LIN {X 0,Y 737.28,Z 922.886,A -85,B 0,C 180,E1 34854.05,E2 34854.05} C_VEL
LIN {X 0,Y 736.992,Z 943.234,A -85,B 0,C 180,E1 34852.747,E2 34852.747} C_VEL
LIN {X 0,Y 736.792,Z 961.106,A -85,B 0,C 180,E1 34851.449,E2 34851.449} C_VEL
LIN {X 0,Y 736.567,Z 978.603,A -85,B 0,C 180,E1 34850.004,E2 34850.004} C_VEL
LIN {X 0,Y 736.424,Z 994.494,A -85,B 0,C 180,E1 34848.525,E2 34848.525} C_VEL
LIN {X 0,Y 736.245,Z 1009.802,A -85,B 0,C 180,E1 34846.896,E2 34846.896} C_VEL
LIN {X 0,Y 736.159,Z 1022.669,A -85,B 0,C 180,E1 34845.342,E2 34845.342} C_VEL
LIN {X 0,Y 736.056,Z 1035.753,A -85,B 0,C 180,E1 34843.512,E2 34843.512} C_VEL
LIN {X 0,Y 735.988,Z 1045.128,A -85,B 0,C 180,E1 34841.993,E2 34841.993} C_VEL
LIN {X 0,Y 735.962,Z 1054.76,A -85,B 0,C 180,E1 34840.173,E2 34840.173} C_VEL
LIN {X 0,Y 735.918,Z 1062.206,A -85,B 0,C 180,E1 34838.438,E2 34838.438} C_VEL
LIN {X 0,Y 735.911,Z 1067.997,A -85,B 0,C 180,E1 34836.789,E2 34836.789} C_VEL
LIN {X 0,Y 735.917,Z 1073.178,A -85,B 0,C 180,E1 34834.832,E2 34834.832} C_VEL
LIN {X 0,Y 735.916,Z 1076.234,A -85,B 0,C 180,E1 34833.115,E2 34833.115} C_VEL
LIN {X 0,Y 735.907,Z 1078.149,A -85,B 0,C 180,E1 34831.246,E2 34831.246} C_VEL
LIN {X 0,Y 735.891,Z 1078.351,A -85,B 0,C 180,E1 34829.455,E2 34829.455} C_VEL
LIN {X 0,Y 735.914,Z 1077.297,A -85,B 0,C 180,E1 34827.742,E2 34827.742} C_VEL
LIN {X 0,Y 735.908,Z 1074.445,A -85,B 0,C 180,E1 34825.792,E2 34825.792} C_VEL
LIN {X 0,Y 735.918,Z 1070.688,A -85,B 0,C 180,E1 34824.151,E2 34824.151} C_VEL
LIN {X 0,Y 735.911,Z 1064.936,A -85,B 0,C 180,E1 34822.27,E2 34822.27} C_VEL
LIN {X 0,Y 735.931,Z 1057.601,A -85,B 0,C 180,E1 34820.459,E2 34820.459} C_VEL
LIN {X 0,Y 735.974,Z 1049.926,A -85,B 0,C 180,E1 34818.877,E2 34818.877} C_VEL
LIN {X 0,Y 736.039,Z 1038.526,A -85,B 0,C 180,E1 34816.914,E2 34816.914} C_VEL
LIN {X 0,Y 736.104,Z 1027.954,A -85,B 0,C 180,E1 34815.365,E2 34815.365} C_VEL
LIN {X 0,Y 736.23,Z 1014.045,A -85,B 0,C 180,E1 34813.591,E2 34813.591} C_VEL
LIN {X 0,Y 736.33,Z 1000.068,A -85,B 0,C 180,E1 34812.046,E2 34812.046} C_VEL
LIN {X 0,Y 736.542,Z 983.248,A -85,B 0,C 180,E1 34810.408,E2 34810.408} C_VEL
LIN {X 0,Y 736.708,Z 966.807,A -85,B 0,C 180,E1 34809.003,E2 34809.003} C_VEL
LIN {X 0,Y 736.965,Z 946.856,A -85,B 0,C 180,E1 34807.505,E2 34807.505} C_VEL
LIN {X 0,Y 737.196,Z 928.356,A -85,B 0,C 180,E1 34806.282,E2 34806.282} C_VEL
LIN {X 0,Y 737.48,Z 906.347,A -85,B 0,C 180,E1 34805.018,E2 34805.018} C_VEL
LIN {X 0,Y 737.719,Z 886.789,A -85,B 0,C 180,E1 34804.037,E2 34804.037} C_VEL
LIN {X 0,Y 738.022,Z 863.387,A -85,B 0,C 180,E1 34803.034,E2 34803.034} C_VEL
LIN {X 0,Y 738.198,Z 843.697,A -85,B 0,C 180,E1 34802.316,E2 34802.316} C_VEL
LIN {X 0,Y 738.494,Z 820.044,A -85,B 0,C 180,E1 34801.595,E2 34801.595} C_VEL
LIN {X 0,Y 738.641,Z 797.319,A -85,B 0,C 180,E1 34801.051,E2 34801.051} C_VEL
LIN {X 0,Y 738.792,Z 776.074,A -85,B 0,C 180,E1 34800.656,E2 34800.656} C_VEL
LIN {X 0,Y 738.933,Z 744.92,A -85,B 0,C 180,E1 34800.262,E2 34800.262} C_VEL
LIN {X 0,Y 739.5,Z 493.491,A -85,B 0,C 180,E1 34797.493,E2 34797.493} C_VEL
LIN {X 0,Y 739.604,Z 381.804,A -85,B 0,C 180,E1 34796.229,E2 34796.229} C_VEL
LIN {X 0,Y 738.409,Z 376.685,A -85,B 0,C 180,E1 34796.09,E2 34796.09} C_VEL
LIN {X 0,Y 738.712,Z 341.298,A -85,B 0,C 180,E1 34793.646,E2 34793.646} C_VEL
LIN {X 0,Y 738.481,Z 336.305,A -85,B 0,C 180,E1 34793.28,E2 34793.28} C_VEL
LIN {X 0,Y 736.045,Z 329.548,A -85,B 0,C 180,E1 34792.627,E2 34792.627} C_VEL
LIN {X 0,Y 736.024,Z 329.546,A -85,B 0,C 180,E1 34790.118,E2 34790.118} C_VEL
LIN {X 0,Y 736.063,Z 329.539,A -85,B 0,C 180,E1 34787.53,E2 34787.53} C_VEL
LIN {X 0,Y 736.046,Z 329.544,A -85,B 0,C 180,E1 34784.505,E2 34784.505} C_VEL
LIN {X 0,Y 736.024,Z 329.541,A -85,B 0,C 180,E1 34781.943,E2 34781.943} C_VEL
LIN {X 0,Y 736.082,Z 329.536,A -85,B 0,C 180,E1 34779.26,E2 34779.26} C_VEL
LIN {X 0,Y 736.042,Z 329.543,A -85,B 0,C 180,E1 34776.32,E2 34776.32} C_VEL
LIN {X 0,Y 736.026,Z 329.539,A -85,B 0,C 180,E1 34773.754,E2 34773.754} C_VEL
LIN {X 0,Y 736.099,Z 329.536,A -85,B 0,C 180,E1 34770.986,E2 34770.986} C_VEL
LIN {X 0,Y 736.038,Z 329.54,A -85,B 0,C 180,E1 34768.125,E2 34768.125} C_VEL
LIN {X 0,Y 736.028,Z 329.539,A -85,B 0,C 180,E1 34765.595,E2 34765.595} C_VEL
LIN {X 0,Y 736.1,Z 329.534,A -85,B 0,C 180,E1 34762.861,E2 34762.861} C_VEL
LIN {X 0,Y 736.034,Z 329.54,A -85,B 0,C 180,E1 34759.937,E2 34759.937} C_VEL
LIN {X 0,Y 736.031,Z 329.539,A -85,B 0,C 180,E1 34757.39,E2 34757.39} C_VEL
LIN {X 0,Y 736.099,Z 329.539,A -85,B 0,C 180,E1 34754.554,E2 34754.554} C_VEL
LIN {X 0,Y 736.033,Z 329.541,A -85,B 0,C 180,E1 34751.758,E2 34751.758} C_VEL
LIN {X 0,Y 736.033,Z 329.536,A -85,B 0,C 180,E1 34749.224,E2 34749.224} C_VEL
LIN {X 0,Y 736.1,Z 329.54,A -85,B 0,C 180,E1 34746.395,E2 34746.395} C_VEL
LIN {X 0,Y 736.032,Z 329.54,A -85,B 0,C 180,E1 34743.583,E2 34743.583} C_VEL
LIN {X 0,Y 736.037,Z 329.538,A -85,B 0,C 180,E1 34741.029,E2 34741.029} C_VEL
LIN {X 0,Y 736.097,Z 329.54,A -85,B 0,C 180,E1 34738.132,E2 34738.132} C_VEL
LIN {X 0,Y 736.03,Z 329.54,A -85,B 0,C 180,E1 34735.403,E2 34735.403} C_VEL
LIN {X 0,Y 736.037,Z 329.537,A -85,B 0,C 180,E1 34732.899,E2 34732.899} C_VEL
LIN {X 0,Y 736.097,Z 329.543,A -85,B 0,C 180,E1 34729.987,E2 34729.987} C_VEL
LIN {X 0,Y 736.028,Z 329.537,A -85,B 0,C 180,E1 34729.196,E2 34729.196} C_VEL
LIN {X 0,Y 735.028,Z 329.666,A -85,B 0,C 180,E1 34728.597,E2 34728.597} C_VEL
LIN {X 0,Y 728.625,Z 330.464,A -85,B 0,C 180,E1 34726.917,E2 34726.917} C_VEL
LIN {X 0,Y 728.13,Z 330.525,A -85,B 0,C 180,E1 34726.481,E2 34726.481} C_VEL
LIN {X 0,Y 728.109,Z 330.53,A -85,B 0,C 180,E1 34723.444,E2 34723.444} C_VEL
LIN {X 0,Y 728.092,Z 330.528,A -85,B 0,C 180,E1 34720.839,E2 34720.839} C_VEL
LIN {X 0,Y 728.159,Z 330.523,A -85,B 0,C 180,E1 34718.068,E2 34718.068} C_VEL
LIN {X 0,Y 728.097,Z 330.527,A -85,B 0,C 180,E1 34715.151,E2 34715.151} C_VEL
LIN {X 0,Y 728.096,Z 330.528,A -85,B 0,C 180,E1 34712.609,E2 34712.609} C_VEL
LIN {X 0,Y 728.16,Z 330.527,A -85,B 0,C 180,E1 34709.738,E2 34709.738} C_VEL
LIN {X 0,Y 728.093,Z 330.527,A -85,B 0,C 180,E1 34706.899,E2 34706.899} C_VEL
LIN {X 0,Y 728.11,Z 330.527,A -85,B 0,C 180,E1 34704.293,E2 34704.293} C_VEL
LIN {X 0,Y 728.13,Z 330.532,A -85,B 0,C 180,E1 34701.23,E2 34701.23} C_VEL
LIN {X 0,Y 728.092,Z 330.53,A -85,B 0,C 180,E1 34698.552,E2 34698.552} C_VEL
LIN {X 0,Y 728.156,Z 330.519,A -85,B 0,C 180,E1 34695.767,E2 34695.767} C_VEL
LIN {X 0,Y 728.104,Z 330.53,A -85,B 0,C 180,E1 34692.826,E2 34692.826} C_VEL
LIN {X 0,Y 728.099,Z 330.529,A -85,B 0,C 180,E1 34690.222,E2 34690.222} C_VEL
LIN {X 0,Y 728.161,Z 330.532,A -85,B 0,C 180,E1 34687.338,E2 34687.338} C_VEL
LIN {X 0,Y 728.095,Z 330.536,A -85,B 0,C 180,E1 34684.515,E2 34684.515} C_VEL
LIN {X 0,Y 728.157,Z 330.634,A -85,B 0,C 180,E1 34683.663,E2 34683.663} C_VEL
LIN {X 0,Y 731.175,Z 340.419,A -85,B 0,C 180,E1 34682.752,E2 34682.752} C_VEL
LIN {X 0,Y 731.211,Z 347.847,A -85,B 0,C 180,E1 34682.212,E2 34682.212} C_VEL
LIN {X 0,Y 733.078,Z 355.743,A -85,B 0,C 180,E1 34682.022,E2 34682.022} C_VEL
LIN {X 0,Y 732.35,Z 591.479,A -85,B 0,C 180,E1 34679.367,E2 34679.367} C_VEL
LIN {X 0,Y 731.891,Z 736.674,A -85,B 0,C 180,E1 34677.744,E2 34677.744} C_VEL
LIN {X 0,Y 731.635,Z 762.056,A -85,B 0,C 180,E1 34677.321,E2 34677.321} C_VEL
LIN {X 0,Y 731.419,Z 783.723,A -85,B 0,C 180,E1 34676.824,E2 34676.824} C_VEL
LIN {X 0,Y 731.163,Z 806.722,A -85,B 0,C 180,E1 34676.17,E2 34676.17} C_VEL
LIN {X 0,Y 730.791,Z 829.655,A -85,B 0,C 180,E1 34675.357,E2 34675.357} C_VEL
LIN {X 0,Y 730.482,Z 852.136,A -85,B 0,C 180,E1 34674.417,E2 34674.417} C_VEL
LIN {X 0,Y 730.067,Z 873.566,A -85,B 0,C 180,E1 34673.359,E2 34673.359} C_VEL
LIN {X 0,Y 729.754,Z 893.71,A -85,B 0,C 180,E1 34672.22,E2 34672.22} C_VEL
LIN {X 0,Y 729.388,Z 913.66,A -85,B 0,C 180,E1 34670.923,E2 34670.923} C_VEL
LIN {X 0,Y 729.096,Z 932.306,A -85,B 0,C 180,E1 34669.55,E2 34669.55} C_VEL
LIN {X 0,Y 728.785,Z 949.92,A -85,B 0,C 180,E1 34668.063,E2 34668.063} C_VEL
LIN {X 0,Y 728.585,Z 966.339,A -85,B 0,C 180,E1 34666.504,E2 34666.504} C_VEL
LIN {X 0,Y 728.356,Z 981.216,A -85,B 0,C 180,E1 34664.875,E2 34664.875} C_VEL
LIN {X 0,Y 728.216,Z 994.942,A -85,B 0,C 180,E1 34663.175,E2 34663.175} C_VEL
LIN {X 0,Y 728.096,Z 1006.602,A -85,B 0,C 180,E1 34661.486,E2 34661.486} C_VEL
LIN {X 0,Y 728.022,Z 1016.711,A -85,B 0,C 180,E1 34659.806,E2 34659.806} C_VEL
LIN {X 0,Y 727.951,Z 1026.298,A -85,B 0,C 180,E1 34657.895,E2 34657.895} C_VEL
LIN {X 0,Y 727.932,Z 1032.884,A -85,B 0,C 180,E1 34656.309,E2 34656.309} C_VEL
LIN {X 0,Y 727.913,Z 1039.273,A -85,B 0,C 180,E1 34654.412,E2 34654.412} C_VEL
LIN {X 0,Y 727.914,Z 1043.665,A -85,B 0,C 180,E1 34652.598,E2 34652.598} C_VEL
LIN {X 0,Y 727.906,Z 1046.575,A -85,B 0,C 180,E1 34650.866,E2 34650.866} C_VEL
LIN {X 0,Y 727.904,Z 1048.262,A -85,B 0,C 180,E1 34648.819,E2 34648.819} C_VEL
LIN {X 0,Y 727.9,Z 1048.283,A -85,B 0,C 180,E1 34647.165,E2 34647.165} C_VEL
LIN {X 0,Y 727.897,Z 1046.788,A -85,B 0,C 180,E1 34645.193,E2 34645.193} C_VEL
LIN {X 0,Y 727.916,Z 1043.949,A -85,B 0,C 180,E1 34643.453,E2 34643.453} C_VEL
LIN {X 0,Y 727.917,Z 1039.818,A -85,B 0,C 180,E1 34641.707,E2 34641.707} C_VEL
LIN {X 0,Y 727.938,Z 1033.314,A -85,B 0,C 180,E1 34639.714,E2 34639.714} C_VEL
LIN {X 0,Y 727.949,Z 1026.72,A -85,B 0,C 180,E1 34638.11,E2 34638.11} C_VEL
LIN {X 0,Y 728.024,Z 1018.026,A -85,B 0,C 180,E1 34636.336,E2 34636.336} C_VEL
LIN {X 0,Y 728.091,Z 1007.401,A -85,B 0,C 180,E1 34634.549,E2 34634.549} C_VEL
LIN {X 0,Y 728.196,Z 995.974,A -85,B 0,C 180,E1 34632.879,E2 34632.879} C_VEL
LIN {X 0,Y 728.355,Z 982.459,A -85,B 0,C 180,E1 34631.179,E2 34631.179} C_VEL
LIN {X 0,Y 728.531,Z 968.364,A -85,B 0,C 180,E1 34629.62,E2 34629.62} C_VEL
LIN {X 0,Y 728.763,Z 951.659,A -85,B 0,C 180,E1 34628.002,E2 34628.002} C_VEL
LIN {X 0,Y 729.047,Z 934.836,A -85,B 0,C 180,E1 34626.563,E2 34626.563} C_VEL
LIN {X 0,Y 729.341,Z 916.302,A -85,B 0,C 180,E1 34625.172,E2 34625.172} C_VEL
LIN {X 0,Y 729.671,Z 898.222,A -85,B 0,C 180,E1 34623.969,E2 34623.969} C_VEL
LIN {X 0,Y 730.026,Z 877.05,A -85,B 0,C 180,E1 34622.738,E2 34622.738} C_VEL
LIN {X 0,Y 730.364,Z 857.102,A -85,B 0,C 180,E1 34621.726,E2 34621.726} C_VEL
LIN {X 0,Y 730.753,Z 833.775,A -85,B 0,C 180,E1 34620.714,E2 34620.714} C_VEL
LIN {X 0,Y 731.015,Z 812.586,A -85,B 0,C 180,E1 34619.936,E2 34619.936} C_VEL
LIN {X 0,Y 731.403,Z 787.347,A -85,B 0,C 180,E1 34619.179,E2 34619.179} C_VEL
LIN {X 0,Y 731.608,Z 765.993,A -85,B 0,C 180,E1 34618.672,E2 34618.672} C_VEL
LIN {X 0,Y 731.866,Z 742.201,A -85,B 0,C 180,E1 34618.239,E2 34618.239} C_VEL
LIN {X 0,Y 732.018,Z 702.478,A -85,B 0,C 180,E1 34617.769,E2 34617.769} C_VEL
LIN {X 0,Y 732.808,Z 447.857,A -85,B 0,C 180,E1 34614.935,E2 34614.935} C_VEL
LIN {X 0,Y 732.898,Z 354.153,A -85,B 0,C 180,E1 34613.86,E2 34613.86} C_VEL
LIN {X 0,Y 731.135,Z 347.503,A -85,B 0,C 180,E1 34613.689,E2 34613.689} C_VEL
LIN {X 0,Y 731.178,Z 339.723,A -85,B 0,C 180,E1 34613.106,E2 34613.106} C_VEL
LIN {X 0,Y 728.14,Z 330.532,A -85,B 0,C 180,E1 34612.233,E2 34612.233} C_VEL
LIN {X 0,Y 728.09,Z 330.532,A -85,B 0,C 180,E1 34609.536,E2 34609.536} C_VEL
LIN {X 0,Y 728.135,Z 330.533,A -85,B 0,C 180,E1 34606.854,E2 34606.854} C_VEL
LIN {X 0,Y 728.111,Z 330.526,A -85,B 0,C 180,E1 34603.866,E2 34603.866} C_VEL
LIN {X 0,Y 728.09,Z 330.528,A -85,B 0,C 180,E1 34601.306,E2 34601.306} C_VEL
LIN {X 0,Y 728.154,Z 330.532,A -85,B 0,C 180,E1 34598.567,E2 34598.567} C_VEL
LIN {X 0,Y 728.101,Z 330.52,A -85,B 0,C 180,E1 34595.611,E2 34595.611} C_VEL
LIN {X 0,Y 728.094,Z 330.53,A -85,B 0,C 180,E1 34593.038,E2 34593.038} C_VEL
LIN {X 0,Y 728.161,Z 330.528,A -85,B 0,C 180,E1 34590.171,E2 34590.171} C_VEL
LIN {X 0,Y 728.096,Z 330.528,A -85,B 0,C 180,E1 34587.391,E2 34587.391} C_VEL
LIN {X 0,Y 728.098,Z 330.529,A -85,B 0,C 180,E1 34584.805,E2 34584.805} C_VEL
LIN {X 0,Y 728.153,Z 330.523,A -85,B 0,C 180,E1 34581.833,E2 34581.833} C_VEL
LIN {X 0,Y 728.089,Z 330.529,A -85,B 0,C 180,E1 34579.078,E2 34579.078} C_VEL
LIN {X 0,Y 728.121,Z 330.531,A -85,B 0,C 180,E1 34576.433,E2 34576.433} C_VEL
LIN {X 0,Y 728.117,Z 330.525,A -85,B 0,C 180,E1 34573.42,E2 34573.42} C_VEL
LIN {X 0,Y 728.089,Z 330.529,A -85,B 0,C 180,E1 34570.845,E2 34570.845} C_VEL
LIN {X 0,Y 728.149,Z 330.532,A -85,B 0,C 180,E1 34568.08,E2 34568.08} C_VEL
LIN {X 0,Y 728.101,Z 330.526,A -85,B 0,C 180,E1 34565.121,E2 34565.121} C_VEL
LIN {X 0,Y 728.089,Z 330.53,A -85,B 0,C 180,E1 34562.598,E2 34562.598} C_VEL
LIN {X 0,Y 728.163,Z 330.531,A -85,B 0,C 180,E1 34559.764,E2 34559.764} C_VEL
LIN {X 0,Y 728.097,Z 330.525,A -85,B 0,C 180,E1 34556.93,E2 34556.93} C_VEL
LIN {X 0,Y 728.091,Z 330.53,A -85,B 0,C 180,E1 34554.404,E2 34554.404} C_VEL
LIN {X 0,Y 728.162,Z 330.531,A -85,B 0,C 180,E1 34551.63,E2 34551.63} C_VEL
LIN {X 0,Y 728.094,Z 330.525,A -85,B 0,C 180,E1 34548.755,E2 34548.755} C_VEL
LIN {X 0,Y 728.091,Z 330.53,A -85,B 0,C 180,E1 34546.256,E2 34546.256} C_VEL
LIN {X 0,Y 728.16,Z 330.529,A -85,B 0,C 180,E1 34543.404,E2 34543.404} C_VEL
LIN {X 0,Y 728.09,Z 330.525,A -85,B 0,C 180,E1 34540.589,E2 34540.589} C_VEL
LIN {X 0,Y 728.093,Z 330.531,A -85,B 0,C 180,E1 34538.066,E2 34538.066} C_VEL
LIN {X 0,Y 728.162,Z 330.527,A -85,B 0,C 180,E1 34535.185,E2 34535.185} C_VEL
LIN {X 0,Y 728.089,Z 330.527,A -85,B 0,C 180,E1 34532.343,E2 34532.343} C_VEL
LIN {X 0,Y 728.1,Z 330.531,A -85,B 0,C 180,E1 34529.826,E2 34529.826} C_VEL
LIN {X 0,Y 728.146,Z 330.527,A -85,B 0,C 180,E1 34526.87,E2 34526.87} C_VEL
LIN {X 0,Y 728.087,Z 330.53,A -85,B 0,C 180,E1 34524.195,E2 34524.195} C_VEL
LIN {X 0,Y 728.106,Z 330.531,A -85,B 0,C 180,E1 34521.631,E2 34521.631} C_VEL
LIN {X 0,Y 728.122,Z 330.527,A -85,B 0,C 180,E1 34518.554,E2 34518.554} C_VEL
LIN {X 0,Y 728.086,Z 330.53,A -85,B 0,C 180,E1 34515.91,E2 34515.91} C_VEL
LIN {X 0,Y 728.131,Z 330.534,A -85,B 0,C 180,E1 34513.255,E2 34513.255} C_VEL
LIN {X 0,Y 728.108,Z 330.531,A -85,B 0,C 180,E1 34510.302,E2 34510.302} C_VEL
LIN {X 0,Y 728.095,Z 330.601,A -85,B 0,C 180,E1 34507.747,E2 34507.747} C_VEL
LIN {X 0,Y 731.737,Z 340.721,A -85,B 0,C 180,E1 34506.798,E2 34506.798} C_VEL
LIN {X 0,Y 731.312,Z 376.071,A -85,B 0,C 180,E1 34504.328,E2 34504.328} C_VEL
LIN {X 0,Y 731.483,Z 377.843,A -85,B 0,C 180,E1 34504.243,E2 34504.243} C_VEL
LIN {X 0,Y 733.119,Z 385.204,A -85,B 0,C 180,E1 34504.071,E2 34504.071} C_VEL
LIN {X 0,Y 732.283,Z 644.202,A -85,B 0,C 180,E1 34501.16,E2 34501.16} C_VEL
LIN {X 0,Y 731.89,Z 766.852,A -85,B 0,C 180,E1 34499.787,E2 34499.787} C_VEL
LIN {X 0,Y 731.63,Z 792.379,A -85,B 0,C 180,E1 34499.36,E2 34499.36} C_VEL
LIN {X 0,Y 731.417,Z 813.903,A -85,B 0,C 180,E1 34498.865,E2 34498.865} C_VEL
LIN {X 0,Y 731.153,Z 837.29,A -85,B 0,C 180,E1 34498.196,E2 34498.196} C_VEL
LIN {X 0,Y 730.784,Z 860.276,A -85,B 0,C 180,E1 34497.378,E2 34497.378} C_VEL
LIN {X 0,Y 730.482,Z 882.073,A -85,B 0,C 180,E1 34496.465,E2 34496.465} C_VEL
LIN {X 0,Y 730.059,Z 903.946,A -85,B 0,C 180,E1 34495.384,E2 34495.384} C_VEL
LIN {X 0,Y 729.749,Z 924.343,A -85,B 0,C 180,E1 34494.228,E2 34494.228} C_VEL
LIN {X 0,Y 729.364,Z 944.443,A -85,B 0,C 180,E1 34492.913,E2 34492.913} C_VEL
LIN {X 0,Y 729.086,Z 963.251,A -85,B 0,C 180,E1 34491.522,E2 34491.522} C_VEL
LIN {X 0,Y 728.782,Z 980.461,A -85,B 0,C 180,E1 34490.06,E2 34490.06} C_VEL
LIN {X 0,Y 728.57,Z 996.962,A -85,B 0,C 180,E1 34488.483,E2 34488.483} C_VEL
LIN {X 0,Y 728.358,Z 1011.447,A -85,B 0,C 180,E1 34486.893,E2 34486.893} C_VEL
LIN {X 0,Y 728.222,Z 1025.058,A -85,B 0,C 180,E1 34485.204,E2 34485.204} C_VEL
LIN {X 0,Y 728.102,Z 1036.794,A -85,B 0,C 180,E1 34483.501,E2 34483.501} C_VEL
LIN {X 0,Y 728.013,Z 1046.95,A -85,B 0,C 180,E1 34481.809,E2 34481.809} C_VEL
LIN {X 0,Y 727.951,Z 1056.181,A -85,B 0,C 180,E1 34479.966,E2 34479.966} C_VEL
LIN {X 0,Y 727.929,Z 1062.815,A -85,B 0,C 180,E1 34478.372,E2 34478.372} C_VEL
LIN {X 0,Y 727.905,Z 1069.245,A -85,B 0,C 180,E1 34476.468,E2 34476.468} C_VEL
LIN {X 0,Y 727.917,Z 1073.654,A -85,B 0,C 180,E1 34474.649,E2 34474.649} C_VEL
LIN {X 0,Y 727.911,Z 1076.572,A -85,B 0,C 180,E1 34472.913,E2 34472.913} C_VEL
LIN {X 0,Y 727.905,Z 1078.262,A -85,B 0,C 180,E1 34470.866,E2 34470.866} C_VEL
LIN {X 0,Y 727.899,Z 1078.284,A -85,B 0,C 180,E1 34469.213,E2 34469.213} C_VEL
LIN {X 0,Y 727.906,Z 1076.796,A -85,B 0,C 180,E1 34467.244,E2 34467.244} C_VEL
LIN {X 0,Y 727.913,Z 1073.813,A -85,B 0,C 180,E1 34465.43,E2 34465.43} C_VEL
LIN {X 0,Y 727.907,Z 1069.451,A -85,B 0,C 180,E1 34463.612,E2 34463.612} C_VEL
LIN {X 0,Y 727.935,Z 1063.118,A -85,B 0,C 180,E1 34461.707,E2 34461.707} C_VEL
LIN {X 0,Y 727.947,Z 1056.536,A -85,B 0,C 180,E1 34460.114,E2 34460.114} C_VEL
LIN {X 0,Y 728.016,Z 1047.41,A -85,B 0,C 180,E1 34458.272,E2 34458.272} C_VEL
LIN {X 0,Y 728.099,Z 1037.315,A -85,B 0,C 180,E1 34456.58,E2 34456.58} C_VEL
LIN {X 0,Y 728.214,Z 1025.489,A -85,B 0,C 180,E1 34454.856,E2 34454.856} C_VEL
LIN {X 0,Y 728.358,Z 1011.926,A -85,B 0,C 180,E1 34453.162,E2 34453.162} C_VEL
LIN {X 0,Y 728.547,Z 997.739,A -85,B 0,C 180,E1 34451.599,E2 34451.599} C_VEL
LIN {X 0,Y 728.773,Z 981.391,A -85,B 0,C 180,E1 34450.024,E2 34450.024} C_VEL
LIN {X 0,Y 729.064,Z 964.272,A -85,B 0,C 180,E1 34448.562,E2 34448.562} C_VEL
LIN {X 0,Y 729.347,Z 945.65,A -85,B 0,C 180,E1 34447.171,E2 34447.171} C_VEL
LIN {X 0,Y 729.72,Z 926.427,A -85,B 0,C 180,E1 34445.9,E2 34445.9} C_VEL
LIN {X 0,Y 730.042,Z 905.214,A -85,B 0,C 180,E1 34444.684,E2 34444.684} C_VEL
LIN {X 0,Y 730.442,Z 884.085,A -85,B 0,C 180,E1 34443.628,E2 34443.628} C_VEL
LIN {X 0,Y 730.773,Z 861.599,A -85,B 0,C 180,E1 34442.674,E2 34442.674} C_VEL
LIN {X 0,Y 731.067,Z 840.358,A -85,B 0,C 180,E1 34441.907,E2 34441.907} C_VEL
LIN {X 0,Y 731.41,Z 815.372,A -85,B 0,C 180,E1 34441.173,E2 34441.173} C_VEL
LIN {X 0,Y 731.614,Z 794.548,A -85,B 0,C 180,E1 34440.686,E2 34440.686} C_VEL
LIN {X 0,Y 731.882,Z 769.639,A -85,B 0,C 180,E1 34440.249,E2 34440.249} C_VEL
LIN {X 0,Y 732.058,Z 720.307,A -85,B 0,C 180,E1 34439.68,E2 34439.68} C_VEL
LIN {X 0,Y 732.828,Z 469.086,A -85,B 0,C 180,E1 34436.881,E2 34436.881} C_VEL
LIN {X 0,Y 732.922,Z 383.497,A -85,B 0,C 180,E1 34435.899,E2 34435.899} C_VEL
LIN {X 0,Y 731.303,Z 376.685,A -85,B 0,C 180,E1 34435.715,E2 34435.715} C_VEL
LIN {X 0,Y 731.729,Z 341.21,A -85,B 0,C 180,E1 34433.236,E2 34433.236} C_VEL
LIN {X 0,Y 730.55,Z 337.116,A -85,B 0,C 180,E1 34432.873,E2 34432.873} C_VEL
LIN {X 0,Y 728.085,Z 330.536,A -85,B 0,C 180,E1 34432.23,E2 34432.23} C_VEL
LIN {X 0,Y 728.114,Z 330.534,A -85,B 0,C 180,E1 34429.655,E2 34429.655} C_VEL
LIN {X 0,Y 728.114,Z 330.534,A -85,B 0,C 180,E1 34426.59,E2 34426.59} C_VEL
LIN {X 0,Y 728.085,Z 330.531,A -85,B 0,C 180,E1 34424.019,E2 34424.019} C_VEL
LIN {X 0,Y 728.141,Z 330.527,A -85,B 0,C 180,E1 34421.31,E2 34421.31} C_VEL
LIN {X 0,Y 728.104,Z 330.531,A -85,B 0,C 180,E1 34418.359,E2 34418.359} C_VEL
LIN {X 0,Y 728.087,Z 330.529,A -85,B 0,C 180,E1 34415.805,E2 34415.805} C_VEL
LIN {X 0,Y 728.157,Z 330.525,A -85,B 0,C 180,E1 34413.035,E2 34413.035} C_VEL
LIN {X 0,Y 728.096,Z 330.53,A -85,B 0,C 180,E1 34410.097,E2 34410.097} C_VEL
LIN {X 0,Y 728.091,Z 330.526,A -85,B 0,C 180,E1 34407.568,E2 34407.568} C_VEL
LIN {X 0,Y 728.162,Z 330.53,A -85,B 0,C 180,E1 34404.673,E2 34404.673} C_VEL
LIN {X 0,Y 728.092,Z 330.531,A -85,B 0,C 180,E1 34401.934,E2 34401.934} C_VEL
LIN {X 0,Y 728.091,Z 330.526,A -85,B 0,C 180,E1 34399.411,E2 34399.411} C_VEL
LIN {X 0,Y 728.161,Z 330.53,A -85,B 0,C 180,E1 34396.514,E2 34396.514} C_VEL
LIN {X 0,Y 728.092,Z 330.529,A -85,B 0,C 180,E1 34393.744,E2 34393.744} C_VEL
LIN {X 0,Y 728.094,Z 330.528,A -85,B 0,C 180,E1 34391.245,E2 34391.245} C_VEL
LIN {X 0,Y 728.162,Z 330.527,A -85,B 0,C 180,E1 34388.37,E2 34388.37} C_VEL
LIN {X 0,Y 728.092,Z 330.528,A -85,B 0,C 180,E1 34385.596,E2 34385.596} C_VEL
LIN {X 0,Y 728.098,Z 330.526,A -85,B 0,C 180,E1 34383.07,E2 34383.07} C_VEL
LIN {X 0,Y 728.161,Z 330.53,A -85,B 0,C 180,E1 34380.157,E2 34380.157} C_VEL
LIN {X 0,Y 728.091,Z 330.53,A -85,B 0,C 180,E1 34377.402,E2 34377.402} C_VEL
LIN {X 0,Y 728.108,Z 330.525,A -85,B 0,C 180,E1 34374.8,E2 34374.8} C_VEL
LIN {X 0,Y 728.133,Z 330.533,A -85,B 0,C 180,E1 34371.789,E2 34371.789} C_VEL
LIN {X 0,Y 728.089,Z 330.525,A -85,B 0,C 180,E1 34369.086,E2 34369.086} C_VEL
LIN {X 0,Y 728.13,Z 330.525,A -85,B 0,C 180,E1 34366.481,E2 34366.481} C_VEL
LIN {X 0,Y 727.195,Z 330.653,A -85,B 0,C 180,E1 34365.875,E2 34365.875} C_VEL
LIN {X 0,Y 720.682,Z 331.459,A -85,B 0,C 180,E1 34364.134,E2 34364.134} C_VEL
LIN {X 0,Y 720.206,Z 331.518,A -85,B 0,C 180,E1 34363.736,E2 34363.736} C_VEL
LIN {X 0,Y 720.151,Z 331.518,A -85,B 0,C 180,E1 34361.002,E2 34361.002} C_VEL
LIN {X 0,Y 720.193,Z 331.511,A -85,B 0,C 180,E1 34358.327,E2 34358.327} C_VEL
LIN {X 0,Y 720.17,Z 331.516,A -85,B 0,C 180,E1 34355.297,E2 34355.297} C_VEL
LIN {X 0,Y 720.155,Z 331.517,A -85,B 0,C 180,E1 34352.698,E2 34352.698} C_VEL
LIN {X 0,Y 720.222,Z 331.512,A -85,B 0,C 180,E1 34349.873,E2 34349.873} C_VEL
LIN {X 0,Y 720.159,Z 331.516,A -85,B 0,C 180,E1 34346.994,E2 34346.994} C_VEL
LIN {X 0,Y 720.161,Z 331.517,A -85,B 0,C 180,E1 34344.426,E2 34344.426} C_VEL
LIN {X 0,Y 720.218,Z 331.522,A -85,B 0,C 180,E1 34341.438,E2 34341.438} C_VEL
LIN {X 0,Y 720.154,Z 331.52,A -85,B 0,C 180,E1 34338.69,E2 34338.69} C_VEL
LIN {X 0,Y 720.183,Z 331.508,A -85,B 0,C 180,E1 34336.037,E2 34336.037} C_VEL
LIN {X 0,Y 720.178,Z 331.52,A -85,B 0,C 180,E1 34332.972,E2 34332.972} C_VEL
LIN {X 0,Y 720.156,Z 331.519,A -85,B 0,C 180,E1 34330.317,E2 34330.317} C_VEL
LIN {X 0,Y 720.223,Z 331.518,A -85,B 0,C 180,E1 34327.551,E2 34327.551} C_VEL
LIN {X 0,Y 720.161,Z 331.526,A -85,B 0,C 180,E1 34324.602,E2 34324.602} C_VEL
LIN {X 0,Y 720.177,Z 331.614,A -85,B 0,C 180,E1 34324.044,E2 34324.044} C_VEL
LIN {X 0,Y 724.011,Z 342.788,A -85,B 0,C 180,E1 34322.965,E2 34322.965} C_VEL
LIN {X 0,Y 724.098,Z 347.958,A -85,B 0,C 180,E1 34322.595,E2 34322.595} C_VEL
LIN {X 0,Y 726.437,Z 357.404,A -85,B 0,C 180,E1 34322.357,E2 34322.357} C_VEL
LIN {X 0,Y 725.512,Z 593.015,A -85,B 0,C 180,E1 34319.68,E2 34319.68} C_VEL
LIN {X 0,Y 724.937,Z 736.823,A -85,B 0,C 180,E1 34318.057,E2 34318.057} C_VEL
LIN {X 0,Y 724.624,Z 762.352,A -85,B 0,C 180,E1 34317.627,E2 34317.627} C_VEL
LIN {X 0,Y 724.346,Z 784.069,A -85,B 0,C 180,E1 34317.124,E2 34317.124} C_VEL
LIN {X 0,Y 724.009,Z 807.47,A -85,B 0,C 180,E1 34316.448,E2 34316.448} C_VEL
LIN {X 0,Y 723.551,Z 830.3,A -85,B 0,C 180,E1 34315.629,E2 34315.629} C_VEL
LIN {X 0,Y 723.158,Z 852.703,A -85,B 0,C 180,E1 34314.681,E2 34314.681} C_VEL
LIN {X 0,Y 722.63,Z 874.823,A -85,B 0,C 180,E1 34313.571,E2 34313.571} C_VEL
LIN {X 0,Y 722.214,Z 895.894,A -85,B 0,C 180,E1 34312.356,E2 34312.356} C_VEL
LIN {X 0,Y 721.757,Z 915.307,A -85,B 0,C 180,E1 34311.062,E2 34311.062} C_VEL
LIN {X 0,Y 721.375,Z 934.393,A -85,B 0,C 180,E1 34309.623,E2 34309.623} C_VEL
LIN {X 0,Y 721.013,Z 951.109,A -85,B 0,C 180,E1 34308.181,E2 34308.181} C_VEL
LIN {X 0,Y 720.724,Z 968.107,A -85,B 0,C 180,E1 34306.523,E2 34306.523} C_VEL
LIN {X 0,Y 720.471,Z 982.124,A -85,B 0,C 180,E1 34304.959,E2 34304.959} C_VEL
LIN {X 0,Y 720.277,Z 996.262,A -85,B 0,C 180,E1 34303.16,E2 34303.16} C_VEL
LIN {X 0,Y 720.145,Z 1007.27,A -85,B 0,C 180,E1 34301.533,E2 34301.533} C_VEL
LIN {X 0,Y 720.051,Z 1018.192,A -85,B 0,C 180,E1 34299.673,E2 34299.673} C_VEL
LIN {X 0,Y 719.965,Z 1026.754,A -85,B 0,C 180,E1 34297.903,E2 34297.903} C_VEL
LIN {X 0,Y 719.945,Z 1033.577,A -85,B 0,C 180,E1 34296.219,E2 34296.219} C_VEL
LIN {X 0,Y 719.92,Z 1039.949,A -85,B 0,C 180,E1 34294.221,E2 34294.221} C_VEL
LIN {X 0,Y 719.916,Z 1044.027,A -85,B 0,C 180,E1 34292.468,E2 34292.468} C_VEL
LIN {X 0,Y 719.896,Z 1047.044,A -85,B 0,C 180,E1 34290.557,E2 34290.557} C_VEL
LIN {X 0,Y 719.893,Z 1048.313,A -85,B 0,C 180,E1 34288.647,E2 34288.647} C_VEL
LIN {X 0,Y 719.911,Z 1048.21,A -85,B 0,C 180,E1 34286.895,E2 34286.895} C_VEL
LIN {X 0,Y 719.913,Z 1046.418,A -85,B 0,C 180,E1 34284.9,E2 34284.9} C_VEL
LIN {X 0,Y 719.909,Z 1043.586,A -85,B 0,C 180,E1 34283.22,E2 34283.22} C_VEL
LIN {X 0,Y 719.918,Z 1038.879,A -85,B 0,C 180,E1 34281.293,E2 34281.293} C_VEL
LIN {X 0,Y 719.933,Z 1032.921,A -85,B 0,C 180,E1 34279.517,E2 34279.517} C_VEL
LIN {X 0,Y 719.978,Z 1026.19,A -85,B 0,C 180,E1 34277.879,E2 34277.879} C_VEL
LIN {X 0,Y 720.061,Z 1016.044,A -85,B 0,C 180,E1 34275.854,E2 34275.854} C_VEL
LIN {X 0,Y 720.162,Z 1006.099,A -85,B 0,C 180,E1 34274.193,E2 34274.193} C_VEL
LIN {X 0,Y 720.325,Z 993.579,A -85,B 0,C 180,E1 34272.386,E2 34272.386} C_VEL
LIN {X 0,Y 720.485,Z 980.819,A -85,B 0,C 180,E1 34270.797,E2 34270.797} C_VEL
LIN {X 0,Y 720.775,Z 965.502,A -85,B 0,C 180,E1 34269.113,E2 34269.113} C_VEL
LIN {X 0,Y 721.067,Z 949.122,A -85,B 0,C 180,E1 34267.549,E2 34267.549} C_VEL
LIN {X 0,Y 721.435,Z 931.29,A -85,B 0,C 180,E1 34266.041,E2 34266.041} C_VEL
LIN {X 0,Y 721.816,Z 913.167,A -85,B 0,C 180,E1 34264.697,E2 34264.697} C_VEL
LIN {X 0,Y 722.27,Z 891.782,A -85,B 0,C 180,E1 34263.306,E2 34263.306} C_VEL
LIN {X 0,Y 722.701,Z 872.392,A -85,B 0,C 180,E1 34262.209,E2 34262.209} C_VEL
LIN {X 0,Y 723.201,Z 848.869,A -85,B 0,C 180,E1 34261.059,E2 34261.059} C_VEL
LIN {X 0,Y 723.594,Z 828.32,A -85,B 0,C 180,E1 34260.204,E2 34260.204} C_VEL
LIN {X 0,Y 724.064,Z 803.979,A -85,B 0,C 180,E1 34259.354,E2 34259.354} C_VEL
LIN {X 0,Y 724.363,Z 781.807,A -85,B 0,C 180,E1 34258.727,E2 34258.727} C_VEL
LIN {X 0,Y 724.745,Z 757.551,A -85,B 0,C 180,E1 34258.187,E2 34258.187} C_VEL
LIN {X 0,Y 724.949,Z 734.194,A -85,B 0,C 180,E1 34257.818,E2 34257.818} C_VEL
LIN {X 0,Y 725.996,Z 471.715,A -85,B 0,C 180,E1 34254.861,E2 34254.861} C_VEL
LIN {X 0,Y 726.255,Z 355.961,A -85,B 0,C 180,E1 34253.526,E2 34253.526} C_VEL
LIN {X 0,Y 723.986,Z 347.403,A -85,B 0,C 180,E1 34253.295,E2 34253.295} C_VEL
LIN {X 0,Y 723.878,Z 342.446,A -85,B 0,C 180,E1 34252.911,E2 34252.911} C_VEL
LIN {X 0,Y 720.162,Z 331.525,A -85,B 0,C 180,E1 34251.841,E2 34251.841} C_VEL
LIN {X 0,Y 720.159,Z 331.524,A -85,B 0,C 180,E1 34249.265,E2 34249.265} C_VEL
LIN {X 0,Y 720.222,Z 331.515,A -85,B 0,C 180,E1 34246.329,E2 34246.329} C_VEL
LIN {X 0,Y 720.153,Z 331.517,A -85,B 0,C 180,E1 34243.525,E2 34243.525} C_VEL
LIN {X 0,Y 720.171,Z 331.518,A -85,B 0,C 180,E1 34240.945,E2 34240.945} C_VEL
LIN {X 0,Y 720.182,Z 331.515,A -85,B 0,C 180,E1 34237.855,E2 34237.855} C_VEL
LIN {X 0,Y 720.151,Z 331.51,A -85,B 0,C 180,E1 34235.184,E2 34235.184} C_VEL
LIN {X 0,Y 720.219,Z 331.52,A -85,B 0,C 180,E1 34232.404,E2 34232.404} C_VEL
LIN {X 0,Y 720.16,Z 331.517,A -85,B 0,C 180,E1 34229.478,E2 34229.478} C_VEL
LIN {X 0,Y 720.158,Z 331.519,A -85,B 0,C 180,E1 34226.913,E2 34226.913} C_VEL
LIN {X 0,Y 720.223,Z 331.516,A -85,B 0,C 180,E1 34224.002,E2 34224.002} C_VEL
LIN {X 0,Y 720.153,Z 331.515,A -85,B 0,C 180,E1 34221.161,E2 34221.161} C_VEL
LIN {X 0,Y 720.174,Z 331.521,A -85,B 0,C 180,E1 34218.539,E2 34218.539} C_VEL
LIN {X 0,Y 720.178,Z 331.515,A -85,B 0,C 180,E1 34215.46,E2 34215.46} C_VEL
LIN {X 0,Y 720.151,Z 331.517,A -85,B 0,C 180,E1 34212.836,E2 34212.836} C_VEL
LIN {X 0,Y 720.215,Z 331.519,A -85,B 0,C 180,E1 34210.075,E2 34210.075} C_VEL
LIN {X 0,Y 720.158,Z 331.516,A -85,B 0,C 180,E1 34207.098,E2 34207.098} C_VEL
LIN {X 0,Y 720.157,Z 331.518,A -85,B 0,C 180,E1 34204.516,E2 34204.516} C_VEL
LIN {X 0,Y 720.221,Z 331.513,A -85,B 0,C 180,E1 34201.591,E2 34201.591} C_VEL
LIN {X 0,Y 720.151,Z 331.518,A -85,B 0,C 180,E1 34198.807,E2 34198.807} C_VEL
LIN {X 0,Y 720.171,Z 331.518,A -85,B 0,C 180,E1 34196.179,E2 34196.179} C_VEL
LIN {X 0,Y 720.174,Z 331.512,A -85,B 0,C 180,E1 34193.062,E2 34193.062} C_VEL
LIN {X 0,Y 720.149,Z 331.519,A -85,B 0,C 180,E1 34190.49,E2 34190.49} C_VEL
LIN {X 0,Y 720.21,Z 331.518,A -85,B 0,C 180,E1 34187.736,E2 34187.736} C_VEL
LIN {X 0,Y 720.162,Z 331.513,A -85,B 0,C 180,E1 34184.786,E2 34184.786} C_VEL
LIN {X 0,Y 720.152,Z 331.519,A -85,B 0,C 180,E1 34182.214,E2 34182.214} C_VEL
LIN {X 0,Y 720.223,Z 331.518,A -85,B 0,C 180,E1 34179.344,E2 34179.344} C_VEL
LIN {X 0,Y 720.153,Z 331.514,A -85,B 0,C 180,E1 34176.517,E2 34176.517} C_VEL
LIN {X 0,Y 720.156,Z 331.52,A -85,B 0,C 180,E1 34173.976,E2 34173.976} C_VEL
LIN {X 0,Y 720.219,Z 331.514,A -85,B 0,C 180,E1 34171.002,E2 34171.002} C_VEL
LIN {X 0,Y 720.147,Z 331.518,A -85,B 0,C 180,E1 34168.249,E2 34168.249} C_VEL
LIN {X 0,Y 720.168,Z 331.521,A -85,B 0,C 180,E1 34165.688,E2 34165.688} C_VEL
LIN {X 0,Y 720.178,Z 331.516,A -85,B 0,C 180,E1 34162.576,E2 34162.576} C_VEL
LIN {X 0,Y 720.147,Z 331.52,A -85,B 0,C 180,E1 34159.995,E2 34159.995} C_VEL
LIN {X 0,Y 720.202,Z 331.519,A -85,B 0,C 180,E1 34157.259,E2 34157.259} C_VEL
LIN {X 0,Y 720.163,Z 331.518,A -85,B 0,C 180,E1 34154.297,E2 34154.297} C_VEL
LIN {X 0,Y 720.148,Z 331.521,A -85,B 0,C 180,E1 34151.789,E2 34151.789} C_VEL
LIN {X 0,Y 720.224,Z 331.522,A -85,B 0,C 180,E1 34148.969,E2 34148.969} C_VEL
LIN {X 0,Y 720.178,Z 331.658,A -85,B 0,C 180,E1 34148.158,E2 34148.158} C_VEL
LIN {X 0,Y 724.726,Z 343.938,A -85,B 0,C 180,E1 34146.98,E2 34146.98} C_VEL
LIN {X 0,Y 724.3,Z 377.38,A -85,B 0,C 180,E1 34144.636,E2 34144.636} C_VEL
LIN {X 0,Y 726.479,Z 386.984,A -85,B 0,C 180,E1 34144.405,E2 34144.405} C_VEL
LIN {X 0,Y 725.423,Z 646.459,A -85,B 0,C 180,E1 34141.462,E2 34141.462} C_VEL
LIN {X 0,Y 724.936,Z 767.067,A -85,B 0,C 180,E1 34140.099,E2 34140.099} C_VEL
LIN {X 0,Y 724.615,Z 792.768,A -85,B 0,C 180,E1 34139.664,E2 34139.664} C_VEL
LIN {X 0,Y 724.343,Z 814.337,A -85,B 0,C 180,E1 34139.162,E2 34139.162} C_VEL
LIN {X 0,Y 723.978,Z 838.571,A -85,B 0,C 180,E1 34138.456,E2 34138.456} C_VEL
LIN {X 0,Y 723.547,Z 860.481,A -85,B 0,C 180,E1 34137.667,E2 34137.667} C_VEL
LIN {X 0,Y 723.146,Z 883.179,A -85,B 0,C 180,E1 34136.704,E2 34136.704} C_VEL
LIN {X 0,Y 722.632,Z 904.752,A -85,B 0,C 180,E1 34135.62,E2 34135.62} C_VEL
LIN {X 0,Y 722.216,Z 925.848,A -85,B 0,C 180,E1 34134.404,E2 34134.404} C_VEL
LIN {X 0,Y 721.746,Z 945.564,A -85,B 0,C 180,E1 34133.089,E2 34133.089} C_VEL
LIN {X 0,Y 721.365,Z 964.778,A -85,B 0,C 180,E1 34131.636,E2 34131.636} C_VEL
LIN {X 0,Y 721.012,Z 981.391,A -85,B 0,C 180,E1 34130.201,E2 34130.201} C_VEL
LIN {X 0,Y 720.713,Z 998.517,A -85,B 0,C 180,E1 34128.524,E2 34128.524} C_VEL
LIN {X 0,Y 720.475,Z 1012.01,A -85,B 0,C 180,E1 34127.018,E2 34127.018} C_VEL
LIN {X 0,Y 720.287,Z 1026.218,A -85,B 0,C 180,E1 34125.211,E2 34125.211} C_VEL
LIN {X 0,Y 720.15,Z 1037.315,A -85,B 0,C 180,E1 34123.571,E2 34123.571} C_VEL
LIN {X 0,Y 720.044,Z 1047.962,A -85,B 0,C 180,E1 34121.762,E2 34121.762} C_VEL
LIN {X 0,Y 719.96,Z 1056.892,A -85,B 0,C 180,E1 34119.917,E2 34119.917} C_VEL
LIN {X 0,Y 719.941,Z 1063.423,A -85,B 0,C 180,E1 34118.305,E2 34118.305} C_VEL
LIN {X 0,Y 719.913,Z 1069.864,A -85,B 0,C 180,E1 34116.299,E2 34116.299} C_VEL
LIN {X 0,Y 719.916,Z 1073.813,A -85,B 0,C 180,E1 34114.621,E2 34114.621} C_VEL
LIN {X 0,Y 719.907,Z 1076.797,A -85,B 0,C 180,E1 34112.786,E2 34112.786} C_VEL
LIN {X 0,Y 719.9,Z 1078.284,A -85,B 0,C 180,E1 34110.796,E2 34110.796} C_VEL
LIN {X 0,Y 719.906,Z 1078.262,A -85,B 0,C 180,E1 34109.125,E2 34109.125} C_VEL
LIN {X 0,Y 719.913,Z 1076.572,A -85,B 0,C 180,E1 34107.054,E2 34107.054} C_VEL
LIN {X 0,Y 719.919,Z 1073.654,A -85,B 0,C 180,E1 34105.3,E2 34105.3} C_VEL
LIN {X 0,Y 719.908,Z 1069.015,A -85,B 0,C 180,E1 34103.38,E2 34103.38} C_VEL
LIN {X 0,Y 719.933,Z 1062.815,A -85,B 0,C 180,E1 34101.534,E2 34101.534} C_VEL
LIN {X 0,Y 719.974,Z 1056.182,A -85,B 0,C 180,E1 34099.922,E2 34099.922} C_VEL
LIN {X 0,Y 720.049,Z 1046.492,A -85,B 0,C 180,E1 34097.977,E2 34097.977} C_VEL
LIN {X 0,Y 720.154,Z 1036.797,A -85,B 0,C 180,E1 34096.347,E2 34096.347} C_VEL
LIN {X 0,Y 720.323,Z 1024.443,A -85,B 0,C 180,E1 34094.543,E2 34094.543} C_VEL
LIN {X 0,Y 720.483,Z 1011.22,A -85,B 0,C 180,E1 34092.89,E2 34092.89} C_VEL
LIN {X 0,Y 720.769,Z 996.177,A -85,B 0,C 180,E1 34091.226,E2 34091.226} C_VEL
LIN {X 0,Y 721.055,Z 979.533,A -85,B 0,C 180,E1 34089.631,E2 34089.631} C_VEL
LIN {X 0,Y 721.431,Z 961.605,A -85,B 0,C 180,E1 34088.11,E2 34088.11} C_VEL
LIN {X 0,Y 721.806,Z 943.237,A -85,B 0,C 180,E1 34086.747,E2 34086.747} C_VEL
LIN {X 0,Y 722.274,Z 921.436,A -85,B 0,C 180,E1 34085.33,E2 34085.33} C_VEL
LIN {X 0,Y 722.724,Z 901.528,A -85,B 0,C 180,E1 34084.208,E2 34084.208} C_VEL
LIN {X 0,Y 723.207,Z 878.257,A -85,B 0,C 180,E1 34083.077,E2 34083.077} C_VEL
LIN {X 0,Y 723.622,Z 857.111,A -85,B 0,C 180,E1 34082.202,E2 34082.202} C_VEL
LIN {X 0,Y 724.075,Z 832.965,A -85,B 0,C 180,E1 34081.368,E2 34081.368} C_VEL
LIN {X 0,Y 724.365,Z 811.104,A -85,B 0,C 180,E1 34080.754,E2 34080.754} C_VEL
LIN {X 0,Y 724.75,Z 786.45,A -85,B 0,C 180,E1 34080.213,E2 34080.213} C_VEL
LIN {X 0,Y 724.95,Z 763.827,A -85,B 0,C 180,E1 34079.858,E2 34079.858} C_VEL
LIN {X 0,Y 725.947,Z 508.76,A -85,B 0,C 180,E1 34076.985,E2 34076.985} C_VEL
LIN {X 0,Y 726.325,Z 385.42,A -85,B 0,C 180,E1 34075.569,E2 34075.569} C_VEL
LIN {X 0,Y 724.228,Z 376.685,A -85,B 0,C 180,E1 34075.332,E2 34075.332} C_VEL
LIN {X 0,Y 724.705,Z 343.756,A -85,B 0,C 180,E1 34073.005,E2 34073.005} C_VEL
LIN {X 0,Y 720.163,Z 331.523,A -85,B 0,C 180,E1 34071.818,E2 34071.818} C_VEL
LIN {X 0,Y 720.198,Z 331.524,A -85,B 0,C 180,E1 34068.807,E2 34068.807} C_VEL
LIN {X 0,Y 720.148,Z 331.521,A -85,B 0,C 180,E1 34066.105,E2 34066.105} C_VEL
LIN {X 0,Y 720.193,Z 331.517,A -85,B 0,C 180,E1 34063.412,E2 34063.412} C_VEL
LIN {X 0,Y 720.167,Z 331.519,A -85,B 0,C 180,E1 34060.421,E2 34060.421} C_VEL
LIN {X 0,Y 720.149,Z 331.518,A -85,B 0,C 180,E1 34057.857,E2 34057.857} C_VEL
LIN {X 0,Y 720.216,Z 331.516,A -85,B 0,C 180,E1 34055.083,E2 34055.083} C_VEL
LIN {X 0,Y 720.155,Z 331.519,A -85,B 0,C 180,E1 34052.119,E2 34052.119} C_VEL
LIN {X 0,Y 720.157,Z 331.517,A -85,B 0,C 180,E1 34049.531,E2 34049.531} C_VEL
LIN {X 0,Y 720.218,Z 331.517,A -85,B 0,C 180,E1 34046.61,E2 34046.61} C_VEL
LIN {X 0,Y 720.149,Z 331.515,A -85,B 0,C 180,E1 34043.796,E2 34043.796} C_VEL
LIN {X 0,Y 720.169,Z 331.516,A -85,B 0,C 180,E1 34041.246,E2 34041.246} C_VEL
LIN {X 0,Y 720.188,Z 331.521,A -85,B 0,C 180,E1 34038.203,E2 34038.203} C_VEL
LIN {X 0,Y 720.148,Z 331.517,A -85,B 0,C 180,E1 34035.544,E2 34035.544} C_VEL
LIN {X 0,Y 720.202,Z 331.513,A -85,B 0,C 180,E1 34032.835,E2 34032.835} C_VEL
LIN {X 0,Y 720.164,Z 331.515,A -85,B 0,C 180,E1 34029.833,E2 34029.833} C_VEL
LIN {X 0,Y 720.152,Z 331.517,A -85,B 0,C 180,E1 34027.259,E2 34027.259} C_VEL
LIN {X 0,Y 720.222,Z 331.515,A -85,B 0,C 180,E1 34024.379,E2 34024.379} C_VEL
LIN {X 0,Y 720.153,Z 331.519,A -85,B 0,C 180,E1 34021.512,E2 34021.512} C_VEL
LIN {X 0,Y 720.161,Z 331.511,A -85,B 0,C 180,E1 34018.966,E2 34018.966} C_VEL
LIN {X 0,Y 720.216,Z 331.521,A -85,B 0,C 180,E1 34016.02,E2 34016.02} C_VEL
LIN {X 0,Y 720.152,Z 331.517,A -85,B 0,C 180,E1 34013.302,E2 34013.302} C_VEL
LIN {X 0,Y 720.17,Z 331.516,A -85,B 0,C 180,E1 34010.732,E2 34010.732} C_VEL
LIN {X 0,Y 720.186,Z 331.521,A -85,B 0,C 180,E1 34007.654,E2 34007.654} C_VEL
LIN {X 0,Y 720.15,Z 331.516,A -85,B 0,C 180,E1 34005.034,E2 34005.034} C_VEL
LIN {X 0,Y 720.206,Z 331.518,A -85,B 0,C 180,E1 34003.736,E2 34003.736} C_VEL
LIN {X 0,Y 719.167,Z 331.649,A -85,B 0,C 180,E1 34003.123,E2 34003.123} C_VEL
LIN {X 0,Y 712.739,Z 332.448,A -85,B 0,C 180,E1 34001.407,E2 34001.407} C_VEL
LIN {X 0,Y 712.213,Z 332.507,A -85,B 0,C 180,E1 34000.96,E2 34000.96} C_VEL
LIN {X 0,Y 712.266,Z 332.499,A -85,B 0,C 180,E1 33998.247,E2 33998.247} C_VEL
LIN {X 0,Y 712.229,Z 332.504,A -85,B 0,C 180,E1 33995.269,E2 33995.269} C_VEL
LIN {X 0,Y 712.217,Z 332.506,A -85,B 0,C 180,E1 33992.672,E2 33992.672} C_VEL
LIN {X 0,Y 712.282,Z 332.501,A -85,B 0,C 180,E1 33989.831,E2 33989.831} C_VEL
LIN {X 0,Y 712.217,Z 332.505,A -85,B 0,C 180,E1 33986.944,E2 33986.944} C_VEL
LIN {X 0,Y 712.227,Z 332.505,A -85,B 0,C 180,E1 33984.365,E2 33984.365} C_VEL
LIN {X 0,Y 712.269,Z 332.51,A -85,B 0,C 180,E1 33981.34,E2 33981.34} C_VEL
LIN {X 0,Y 712.215,Z 332.509,A -85,B 0,C 180,E1 33978.605,E2 33978.605} C_VEL
LIN {X 0,Y 712.27,Z 332.495,A -85,B 0,C 180,E1 33975.836,E2 33975.836} C_VEL
LIN {X 0,Y 712.23,Z 332.509,A -85,B 0,C 180,E1 33972.876,E2 33972.876} C_VEL
LIN {X 0,Y 712.222,Z 332.508,A -85,B 0,C 180,E1 33970.225,E2 33970.225} C_VEL
LIN {X 0,Y 712.284,Z 332.51,A -85,B 0,C 180,E1 33967.255,E2 33967.255} C_VEL
LIN {X 0,Y 712.233,Z 332.633,A -85,B 0,C 180,E1 33964.431,E2 33964.431} C_VEL
LIN {X 0,Y 716.874,Z 346.258,A -85,B 0,C 180,E1 33963.097,E2 33963.097} C_VEL
LIN {X 0,Y 717.012,Z 348.148,A -85,B 0,C 180,E1 33962.985,E2 33962.985} C_VEL
LIN {X 0,Y 719.82,Z 359.326,A -85,B 0,C 180,E1 33962.696,E2 33962.696} C_VEL
LIN {X 0,Y 718.694,Z 595.051,A -85,B 0,C 180,E1 33959.993,E2 33959.993} C_VEL
LIN {X 0,Y 718.005,Z 736.964,A -85,B 0,C 180,E1 33958.377,E2 33958.377} C_VEL
LIN {X 0,Y 717.641,Z 762.526,A -85,B 0,C 180,E1 33957.942,E2 33957.942} C_VEL
LIN {X 0,Y 717.294,Z 784.203,A -85,B 0,C 180,E1 33957.436,E2 33957.436} C_VEL
LIN {X 0,Y 716.87,Z 808.198,A -85,B 0,C 180,E1 33956.732,E2 33956.732} C_VEL
LIN {X 0,Y 716.361,Z 829.733,A -85,B 0,C 180,E1 33955.954,E2 33955.954} C_VEL
LIN {X 0,Y 715.863,Z 852.405,A -85,B 0,C 180,E1 33954.989,E2 33954.989} C_VEL
LIN {X 0,Y 715.255,Z 874.42,A -85,B 0,C 180,E1 33953.877,E2 33953.877} C_VEL
LIN {X 0,Y 714.733,Z 895.263,A -85,B 0,C 180,E1 33952.67,E2 33952.67} C_VEL
LIN {X 0,Y 714.192,Z 914.96,A -85,B 0,C 180,E1 33951.347,E2 33951.347} C_VEL
LIN {X 0,Y 713.716,Z 933.972,A -85,B 0,C 180,E1 33949.903,E2 33949.903} C_VEL
LIN {X 0,Y 713.27,Z 951.38,A -85,B 0,C 180,E1 33948.386,E2 33948.386} C_VEL
LIN {X 0,Y 712.899,Z 968.676,A -85,B 0,C 180,E1 33946.673,E2 33946.673} C_VEL
LIN {X 0,Y 712.588,Z 983.029,A -85,B 0,C 180,E1 33945.046,E2 33945.046} C_VEL
LIN {X 0,Y 712.339,Z 997.581,A -85,B 0,C 180,E1 33943.144,E2 33943.144} C_VEL
LIN {X 0,Y 712.188,Z 1008.453,A -85,B 0,C 180,E1 33941.5,E2 33941.5} C_VEL
LIN {X 0,Y 712.068,Z 1019.527,A -85,B 0,C 180,E1 33939.538,E2 33939.538} C_VEL
LIN {X 0,Y 711.974,Z 1027.563,A -85,B 0,C 180,E1 33937.829,E2 33937.829} C_VEL
LIN {X 0,Y 711.944,Z 1034.871,A -85,B 0,C 180,E1 33935.965,E2 33935.965} C_VEL
LIN {X 0,Y 711.926,Z 1040.624,A -85,B 0,C 180,E1 33934.027,E2 33934.027} C_VEL
LIN {X 0,Y 711.916,Z 1044.548,A -85,B 0,C 180,E1 33932.254,E2 33932.254} C_VEL
LIN {X 0,Y 711.919,Z 1047.404,A -85,B 0,C 180,E1 33930.161,E2 33930.161} C_VEL
LIN {X 0,Y 711.89,Z 1048.364,A -85,B 0,C 180,E1 33928.471,E2 33928.471} C_VEL
LIN {X 0,Y 711.901,Z 1048.059,A -85,B 0,C 180,E1 33926.538,E2 33926.538} C_VEL
LIN {X 0,Y 711.906,Z 1046.161,A -85,B 0,C 180,E1 33924.681,E2 33924.681} C_VEL
LIN {X 0,Y 711.921,Z 1043.062,A -85,B 0,C 180,E1 33922.9,E2 33922.9} C_VEL
LIN {X 0,Y 711.935,Z 1037.783,A -85,B 0,C 180,E1 33920.868,E2 33920.868} C_VEL
LIN {X 0,Y 711.938,Z 1032.221,A -85,B 0,C 180,E1 33919.234,E2 33919.234} C_VEL
LIN {X 0,Y 712.017,Z 1024.357,A -85,B 0,C 180,E1 33917.345,E2 33917.345} C_VEL
LIN {X 0,Y 712.112,Z 1014.976,A -85,B 0,C 180,E1 33915.526,E2 33915.526} C_VEL
LIN {X 0,Y 712.25,Z 1004.476,A -85,B 0,C 180,E1 33913.778,E2 33913.778} C_VEL
LIN {X 0,Y 712.441,Z 991.458,A -85,B 0,C 180,E1 33911.931,E2 33911.931} C_VEL
LIN {X 0,Y 712.708,Z 978.141,A -85,B 0,C 180,E1 33910.285,E2 33910.285} C_VEL
LIN {X 0,Y 713.004,Z 962.68,A -85,B 0,C 180,E1 33908.616,E2 33908.616} C_VEL
LIN {X 0,Y 713.401,Z 946.869,A -85,B 0,C 180,E1 33907.111,E2 33907.111} C_VEL
LIN {X 0,Y 713.83,Z 928.46,A -85,B 0,C 180,E1 33905.573,E2 33905.573} C_VEL
LIN {X 0,Y 714.333,Z 910.388,A -85,B 0,C 180,E1 33904.239,E2 33904.239} C_VEL
LIN {X 0,Y 714.844,Z 889.874,A -85,B 0,C 180,E1 33902.916,E2 33902.916} C_VEL
LIN {X 0,Y 715.391,Z 870.255,A -85,B 0,C 180,E1 33901.809,E2 33901.809} C_VEL
LIN {X 0,Y 715.937,Z 847.27,A -85,B 0,C 180,E1 33900.691,E2 33900.691} C_VEL
LIN {X 0,Y 716.445,Z 826.736,A -85,B 0,C 180,E1 33899.839,E2 33899.839} C_VEL
LIN {X 0,Y 716.974,Z 802.732,A -85,B 0,C 180,E1 33899.006,E2 33899.006} C_VEL
LIN {X 0,Y 717.328,Z 781.027,A -85,B 0,C 180,E1 33898.392,E2 33898.392} C_VEL
LIN {X 0,Y 717.788,Z 756.2,A -85,B 0,C 180,E1 33897.845,E2 33897.845} C_VEL
LIN {X 0,Y 718.022,Z 733.611,A -85,B 0,C 180,E1 33897.489,E2 33897.489} C_VEL
LIN {X 0,Y 719.275,Z 474.158,A -85,B 0,C 180,E1 33894.54,E2 33894.54} C_VEL
LIN {X 0,Y 719.66,Z 357.915,A -85,B 0,C 180,E1 33893.189,E2 33893.189} C_VEL
LIN {X 0,Y 716.859,Z 347.284,A -85,B 0,C 180,E1 33892.891,E2 33892.891} C_VEL
LIN {X 0,Y 716.355,Z 344.494,A -85,B 0,C 180,E1 33892.647,E2 33892.647} C_VEL
LIN {X 0,Y 712.215,Z 332.516,A -85,B 0,C 180,E1 33891.44,E2 33891.44} C_VEL
LIN {X 0,Y 712.284,Z 332.508,A -85,B 0,C 180,E1 33888.558,E2 33888.558} C_VEL
LIN {X 0,Y 712.216,Z 332.507,A -85,B 0,C 180,E1 33885.641,E2 33885.641} C_VEL
LIN {X 0,Y 712.233,Z 332.509,A -85,B 0,C 180,E1 33882.994,E2 33882.994} C_VEL
LIN {X 0,Y 712.245,Z 332.502,A -85,B 0,C 180,E1 33879.909,E2 33879.909} C_VEL
LIN {X 0,Y 712.213,Z 332.508,A -85,B 0,C 180,E1 33877.248,E2 33877.248} C_VEL
LIN {X 0,Y 712.278,Z 332.503,A -85,B 0,C 180,E1 33874.453,E2 33874.453} C_VEL
LIN {X 0,Y 712.219,Z 332.503,A -85,B 0,C 180,E1 33871.484,E2 33871.484} C_VEL
LIN {X 0,Y 712.224,Z 332.509,A -85,B 0,C 180,E1 33868.878,E2 33868.878} C_VEL
LIN {X 0,Y 712.272,Z 332.501,A -85,B 0,C 180,E1 33865.886,E2 33865.886} C_VEL
LIN {X 0,Y 712.213,Z 332.507,A -85,B 0,C 180,E1 33863.137,E2 33863.137} C_VEL
LIN {X 0,Y 712.249,Z 332.508,A -85,B 0,C 180,E1 33860.46,E2 33860.46} C_VEL
LIN {X 0,Y 712.23,Z 332.503,A -85,B 0,C 180,E1 33857.399,E2 33857.399} C_VEL
LIN {X 0,Y 712.213,Z 332.508,A -85,B 0,C 180,E1 33854.804,E2 33854.804} C_VEL
LIN {X 0,Y 712.283,Z 332.507,A -85,B 0,C 180,E1 33851.921,E2 33851.921} C_VEL
LIN {X 0,Y 712.216,Z 332.505,A -85,B 0,C 180,E1 33849.047,E2 33849.047} C_VEL
LIN {X 0,Y 712.225,Z 332.509,A -85,B 0,C 180,E1 33846.449,E2 33846.449} C_VEL
LIN {X 0,Y 712.266,Z 332.504,A -85,B 0,C 180,E1 33843.461,E2 33843.461} C_VEL
LIN {X 0,Y 712.21,Z 332.504,A -85,B 0,C 180,E1 33840.724,E2 33840.724} C_VEL
LIN {X 0,Y 712.249,Z 332.511,A -85,B 0,C 180,E1 33838.069,E2 33838.069} C_VEL
LIN {X 0,Y 712.228,Z 332.505,A -85,B 0,C 180,E1 33835.007,E2 33835.007} C_VEL
LIN {X 0,Y 712.211,Z 332.504,A -85,B 0,C 180,E1 33832.417,E2 33832.417} C_VEL
LIN {X 0,Y 712.283,Z 332.504,A -85,B 0,C 180,E1 33829.567,E2 33829.567} C_VEL
LIN {X 0,Y 712.216,Z 332.506,A -85,B 0,C 180,E1 33826.689,E2 33826.689} C_VEL
LIN {X 0,Y 712.221,Z 332.505,A -85,B 0,C 180,E1 33824.086,E2 33824.086} C_VEL
LIN {X 0,Y 712.263,Z 332.499,A -85,B 0,C 180,E1 33821.078,E2 33821.078} C_VEL
LIN {X 0,Y 712.209,Z 332.507,A -85,B 0,C 180,E1 33818.332,E2 33818.332} C_VEL
LIN {X 0,Y 712.252,Z 332.507,A -85,B 0,C 180,E1 33815.657,E2 33815.657} C_VEL
LIN {X 0,Y 712.231,Z 332.503,A -85,B 0,C 180,E1 33812.673,E2 33812.673} C_VEL
LIN {X 0,Y 712.209,Z 332.508,A -85,B 0,C 180,E1 33810.106,E2 33810.106} C_VEL
LIN {X 0,Y 712.28,Z 332.51,A -85,B 0,C 180,E1 33807.285,E2 33807.285} C_VEL
LIN {X 0,Y 712.218,Z 332.507,A -85,B 0,C 180,E1 33804.365,E2 33804.365} C_VEL
LIN {X 0,Y 712.214,Z 332.509,A -85,B 0,C 180,E1 33801.831,E2 33801.831} C_VEL
LIN {X 0,Y 712.283,Z 332.506,A -85,B 0,C 180,E1 33798.923,E2 33798.923} C_VEL
LIN {X 0,Y 712.21,Z 332.508,A -85,B 0,C 180,E1 33796.072,E2 33796.072} C_VEL
LIN {X 0,Y 712.231,Z 332.512,A -85,B 0,C 180,E1 33793.463,E2 33793.463} C_VEL
LIN {X 0,Y 712.234,Z 332.511,A -85,B 0,C 180,E1 33790.33,E2 33790.33} C_VEL
LIN {X 0,Y 712.304,Z 332.749,A -85,B 0,C 180,E1 33788.566,E2 33788.566} C_VEL
LIN {X 0,Y 717.694,Z 347.211,A -85,B 0,C 180,E1 33787.164,E2 33787.164} C_VEL
LIN {X 0,Y 717.276,Z 377.475,A -85,B 0,C 180,E1 33785.024,E2 33785.024} C_VEL
LIN {X 0,Y 719.862,Z 388.77,A -85,B 0,C 180,E1 33784.745,E2 33784.745} C_VEL
LIN {X 0,Y 718.585,Z 648.445,A -85,B 0,C 180,E1 33781.774,E2 33781.774} C_VEL
LIN {X 0,Y 718.004,Z 767.174,A -85,B 0,C 180,E1 33780.419,E2 33780.419} C_VEL
LIN {X 0,Y 717.629,Z 792.895,A -85,B 0,C 180,E1 33779.979,E2 33779.979} C_VEL
LIN {X 0,Y 717.291,Z 814.459,A -85,B 0,C 180,E1 33779.474,E2 33779.474} C_VEL
LIN {X 0,Y 716.861,Z 838.568,A -85,B 0,C 180,E1 33778.765,E2 33778.765} C_VEL
LIN {X 0,Y 716.339,Z 860.486,A -85,B 0,C 180,E1 33777.969,E2 33777.969} C_VEL
LIN {X 0,Y 715.831,Z 883.582,A -85,B 0,C 180,E1 33776.978,E2 33776.978} C_VEL
LIN {X 0,Y 715.246,Z 904.756,A -85,B 0,C 180,E1 33775.904,E2 33775.904} C_VEL
LIN {X 0,Y 714.719,Z 925.755,A -85,B 0,C 180,E1 33774.683,E2 33774.683} C_VEL
LIN {X 0,Y 714.177,Z 945.152,A -85,B 0,C 180,E1 33773.378,E2 33773.378} C_VEL
LIN {X 0,Y 713.724,Z 963.809,A -85,B 0,C 180,E1 33771.962,E2 33771.962} C_VEL
LIN {X 0,Y 713.296,Z 980.462,A -85,B 0,C 180,E1 33770.515,E2 33770.515} C_VEL
LIN {X 0,Y 712.938,Z 996.965,A -85,B 0,C 180,E1 33768.904,E2 33768.904} C_VEL
LIN {X 0,Y 712.623,Z 1011.222,A -85,B 0,C 180,E1 33767.305,E2 33767.305} C_VEL
LIN {X 0,Y 712.408,Z 1025.06,A -85,B 0,C 180,E1 33765.55,E2 33765.55} C_VEL
LIN {X 0,Y 712.209,Z 1036.797,A -85,B 0,C 180,E1 33763.808,E2 33763.808} C_VEL
LIN {X 0,Y 712.082,Z 1046.948,A -85,B 0,C 180,E1 33762.077,E2 33762.077} C_VEL
LIN {X 0,Y 711.99,Z 1056.524,A -85,B 0,C 180,E1 33760.114,E2 33760.114} C_VEL
LIN {X 0,Y 711.94,Z 1063.12,A -85,B 0,C 180,E1 33758.48,E2 33758.48} C_VEL
LIN {X 0,Y 711.909,Z 1069.451,A -85,B 0,C 180,E1 33756.532,E2 33756.532} C_VEL
LIN {X 0,Y 711.918,Z 1073.814,A -85,B 0,C 180,E1 33754.673,E2 33754.673} C_VEL
LIN {X 0,Y 711.908,Z 1076.797,A -85,B 0,C 180,E1 33752.818,E2 33752.818} C_VEL
LIN {X 0,Y 711.901,Z 1078.284,A -85,B 0,C 180,E1 33750.805,E2 33750.805} C_VEL
LIN {X 0,Y 711.906,Z 1078.262,A -85,B 0,C 180,E1 33749.115,E2 33749.115} C_VEL
LIN {X 0,Y 711.914,Z 1076.572,A -85,B 0,C 180,E1 33747.021,E2 33747.021} C_VEL
LIN {X 0,Y 711.919,Z 1073.655,A -85,B 0,C 180,E1 33745.247,E2 33745.247} C_VEL
LIN {X 0,Y 711.914,Z 1069.015,A -85,B 0,C 180,E1 33743.306,E2 33743.306} C_VEL
LIN {X 0,Y 711.938,Z 1062.815,A -85,B 0,C 180,E1 33741.438,E2 33741.438} C_VEL
LIN {X 0,Y 712.001,Z 1056.182,A -85,B 0,C 180,E1 33739.808,E2 33739.808} C_VEL
LIN {X 0,Y 712.095,Z 1046.032,A -85,B 0,C 180,E1 33737.759,E2 33737.759} C_VEL
LIN {X 0,Y 712.214,Z 1036.279,A -85,B 0,C 180,E1 33736.109,E2 33736.109} C_VEL
LIN {X 0,Y 712.423,Z 1023.806,A -85,B 0,C 180,E1 33734.284,E2 33734.284} C_VEL
LIN {X 0,Y 712.64,Z 1010.515,A -85,B 0,C 180,E1 33732.611,E2 33732.611} C_VEL
LIN {X 0,Y 712.961,Z 995.334,A -85,B 0,C 180,E1 33730.927,E2 33730.927} C_VEL
LIN {X 0,Y 713.319,Z 979.534,A -85,B 0,C 180,E1 33729.4,E2 33729.4} C_VEL
LIN {X 0,Y 713.767,Z 961.606,A -85,B 0,C 180,E1 33727.862,E2 33727.862} C_VEL
LIN {X 0,Y 714.239,Z 943.237,A -85,B 0,C 180,E1 33726.485,E2 33726.485} C_VEL
LIN {X 0,Y 714.782,Z 922.166,A -85,B 0,C 180,E1 33725.098,E2 33725.098} C_VEL
LIN {X 0,Y 715.321,Z 902.334,A -85,B 0,C 180,E1 33723.965,E2 33723.965} C_VEL
LIN {X 0,Y 715.904,Z 879.254,A -85,B 0,C 180,E1 33722.825,E2 33722.825} C_VEL
LIN {X 0,Y 716.401,Z 858.239,A -85,B 0,C 180,E1 33721.943,E2 33721.943} C_VEL
LIN {X 0,Y 716.951,Z 834.438,A -85,B 0,C 180,E1 33721.103,E2 33721.103} C_VEL
LIN {X 0,Y 717.314,Z 811.86,A -85,B 0,C 180,E1 33720.458,E2 33720.458} C_VEL
LIN {X 0,Y 717.775,Z 787.537,A -85,B 0,C 180,E1 33719.913,E2 33719.913} C_VEL
LIN {X 0,Y 718.02,Z 764.114,A -85,B 0,C 180,E1 33719.541,E2 33719.541} C_VEL
LIN {X 0,Y 719.22,Z 511.246,A -85,B 0,C 180,E1 33716.666,E2 33716.666} C_VEL
LIN {X 0,Y 719.678,Z 387.124,A -85,B 0,C 180,E1 33715.225,E2 33715.225} C_VEL
LIN {X 0,Y 717.183,Z 376.685,A -85,B 0,C 180,E1 33714.942,E2 33714.942} C_VEL
LIN {X 0,Y 717.695,Z 347.209,A -85,B 0,C 180,E1 33712.836,E2 33712.836} C_VEL
LIN {X 0,Y 712.276,Z 332.509,A -85,B 0,C 180,E1 33711.392,E2 33711.392} C_VEL
LIN {X 0,Y 712.219,Z 332.513,A -85,B 0,C 180,E1 33708.442,E2 33708.442} C_VEL
LIN {X 0,Y 712.214,Z 332.51,A -85,B 0,C 180,E1 33705.866,E2 33705.866} C_VEL
LIN {X 0,Y 712.281,Z 332.51,A -85,B 0,C 180,E1 33702.999,E2 33702.999} C_VEL
LIN {X 0,Y 712.213,Z 332.507,A -85,B 0,C 180,E1 33700.206,E2 33700.206} C_VEL
LIN {X 0,Y 712.219,Z 332.506,A -85,B 0,C 180,E1 33697.64,E2 33697.64} C_VEL
LIN {X 0,Y 712.271,Z 332.507,A -85,B 0,C 180,E1 33694.649,E2 33694.649} C_VEL
LIN {X 0,Y 712.209,Z 332.507,A -85,B 0,C 180,E1 33691.957,E2 33691.957} C_VEL
LIN {X 0,Y 712.234,Z 332.505,A -85,B 0,C 180,E1 33689.331,E2 33689.331} C_VEL
LIN {X 0,Y 712.236,Z 332.51,A -85,B 0,C 180,E1 33686.224,E2 33686.224} C_VEL
LIN {X 0,Y 712.211,Z 332.503,A -85,B 0,C 180,E1 33683.586,E2 33683.586} C_VEL
LIN {X 0,Y 712.282,Z 332.504,A -85,B 0,C 180,E1 33680.785,E2 33680.785} C_VEL
LIN {X 0,Y 712.218,Z 332.508,A -85,B 0,C 180,E1 33677.852,E2 33677.852} C_VEL
LIN {X 0,Y 712.218,Z 332.504,A -85,B 0,C 180,E1 33675.304,E2 33675.304} C_VEL
LIN {X 0,Y 712.282,Z 332.508,A -85,B 0,C 180,E1 33672.403,E2 33672.403} C_VEL
LIN {X 0,Y 712.212,Z 332.503,A -85,B 0,C 180,E1 33669.617,E2 33669.617} C_VEL
LIN {X 0,Y 712.231,Z 332.505,A -85,B 0,C 180,E1 33667,E2 33667} C_VEL
LIN {X 0,Y 712.238,Z 332.508,A -85,B 0,C 180,E1 33663.864,E2 33663.864} C_VEL
LIN {X 0,Y 712.214,Z 332.506,A -85,B 0,C 180,E1 33661.207,E2 33661.207} C_VEL
LIN {X 0,Y 712.283,Z 332.498,A -85,B 0,C 180,E1 33658.391,E2 33658.391} C_VEL
LIN {X 0,Y 712.219,Z 332.506,A -85,B 0,C 180,E1 33655.491,E2 33655.491} C_VEL
LIN {X 0,Y 712.22,Z 332.503,A -85,B 0,C 180,E1 33652.903,E2 33652.903} C_VEL
LIN {X 0,Y 712.28,Z 332.507,A -85,B 0,C 180,E1 33649.975,E2 33649.975} C_VEL
LIN {X 0,Y 712.213,Z 332.507,A -85,B 0,C 180,E1 33647.184,E2 33647.184} C_VEL
LIN {X 0,Y 712.233,Z 332.503,A -85,B 0,C 180,E1 33644.613,E2 33644.613} C_VEL
LIN {X 0,Y 712.242,Z 332.51,A -85,B 0,C 180,E1 33641.502,E2 33641.502} C_VEL
LIN {X 0,Y 712.213,Z 332.507,A -85,B 0,C 180,E1 33640.96,E2 33640.96} C_VEL
LIN {X 0,Y 711.228,Z 332.632,A -85,B 0,C 180,E1 33640.341,E2 33640.341} C_VEL
LIN {X 0,Y 704.842,Z 333.422,A -85,B 0,C 180,E1 33638.605,E2 33638.605} C_VEL
LIN {X 0,Y 704.336,Z 333.488,A -85,B 0,C 180,E1 33638.153,E2 33638.153} C_VEL
LIN {X 0,Y 704.281,Z 333.492,A -85,B 0,C 180,E1 33635.15,E2 33635.15} C_VEL
LIN {X 0,Y 704.286,Z 333.495,A -85,B 0,C 180,E1 33632.522,E2 33632.522} C_VEL
LIN {X 0,Y 704.333,Z 333.498,A -85,B 0,C 180,E1 33629.509,E2 33629.509} C_VEL
LIN {X 0,Y 704.275,Z 333.492,A -85,B 0,C 180,E1 33626.744,E2 33626.744} C_VEL
LIN {X 0,Y 704.328,Z 333.493,A -85,B 0,C 180,E1 33624.004,E2 33624.004} C_VEL
LIN {X 0,Y 704.286,Z 333.497,A -85,B 0,C 180,E1 33620.949,E2 33620.949} C_VEL
LIN {X 0,Y 704.284,Z 333.497,A -85,B 0,C 180,E1 33618.312,E2 33618.312} C_VEL
LIN {X 0,Y 704.338,Z 333.483,A -85,B 0,C 180,E1 33615.335,E2 33615.335} C_VEL
LIN {X 0,Y 704.278,Z 333.495,A -85,B 0,C 180,E1 33612.516,E2 33612.516} C_VEL
LIN {X 0,Y 704.322,Z 333.495,A -85,B 0,C 180,E1 33609.811,E2 33609.811} C_VEL
LIN {X 0,Y 704.296,Z 333.504,A -85,B 0,C 180,E1 33606.801,E2 33606.801} C_VEL
LIN {X 0,Y 704.318,Z 333.634,A -85,B 0,C 180,E1 33604.828,E2 33604.828} C_VEL
LIN {X 0,Y 709.413,Z 347.994,A -85,B 0,C 180,E1 33603.418,E2 33603.418} C_VEL
LIN {X 0,Y 710.976,Z 352.032,A -85,B 0,C 180,E1 33603.28,E2 33603.28} C_VEL
LIN {X 0,Y 713.228,Z 361.214,A -85,B 0,C 180,E1 33603.041,E2 33603.041} C_VEL
LIN {X 0,Y 711.9,Z 596.462,A -85,B 0,C 180,E1 33600.319,E2 33600.319} C_VEL
LIN {X 0,Y 711.095,Z 737.104,A -85,B 0,C 180,E1 33598.702,E2 33598.702} C_VEL
LIN {X 0,Y 710.683,Z 762.688,A -85,B 0,C 180,E1 33598.262,E2 33598.262} C_VEL
LIN {X 0,Y 710.264,Z 784.444,A -85,B 0,C 180,E1 33597.75,E2 33597.75} C_VEL
LIN {X 0,Y 709.748,Z 808.927,A -85,B 0,C 180,E1 33597.022,E2 33597.022} C_VEL
LIN {X 0,Y 709.162,Z 830.486,A -85,B 0,C 180,E1 33596.233,E2 33596.233} C_VEL
LIN {X 0,Y 708.547,Z 853.569,A -85,B 0,C 180,E1 33595.234,E2 33595.234} C_VEL
LIN {X 0,Y 707.876,Z 874.78,A -85,B 0,C 180,E1 33594.148,E2 33594.148} C_VEL
LIN {X 0,Y 707.217,Z 896.311,A -85,B 0,C 180,E1 33592.88,E2 33592.88} C_VEL
LIN {X 0,Y 706.618,Z 915.313,A -85,B 0,C 180,E1 33591.587,E2 33591.587} C_VEL
LIN {X 0,Y 706.049,Z 934.283,A -85,B 0,C 180,E1 33590.127,E2 33590.127} C_VEL
LIN {X 0,Y 705.564,Z 950.732,A -85,B 0,C 180,E1 33588.68,E2 33588.68} C_VEL
LIN {X 0,Y 705.13,Z 967.025,A -85,B 0,C 180,E1 33587.069,E2 33587.069} C_VEL
LIN {X 0,Y 704.75,Z 981.839,A -85,B 0,C 180,E1 33585.386,E2 33585.386} C_VEL
LIN {X 0,Y 704.487,Z 995.453,A -85,B 0,C 180,E1 33583.627,E2 33583.627} C_VEL
LIN {X 0,Y 704.269,Z 1007.058,A -85,B 0,C 180,E1 33581.88,E2 33581.88} C_VEL
LIN {X 0,Y 704.119,Z 1017.561,A -85,B 0,C 180,E1 33580.059,E2 33580.059} C_VEL
LIN {X 0,Y 704.013,Z 1026.732,A -85,B 0,C 180,E1 33578.136,E2 33578.136} C_VEL
LIN {X 0,Y 703.947,Z 1033.449,A -85,B 0,C 180,E1 33576.443,E2 33576.443} C_VEL
LIN {X 0,Y 703.921,Z 1040.067,A -85,B 0,C 180,E1 33574.318,E2 33574.318} C_VEL
LIN {X 0,Y 703.915,Z 1043.96,A -85,B 0,C 180,E1 33572.605,E2 33572.605} C_VEL
LIN {X 0,Y 703.899,Z 1046.897,A -85,B 0,C 180,E1 33570.733,E2 33570.733} C_VEL
LIN {X 0,Y 703.9,Z 1048.281,A -85,B 0,C 180,E1 33568.779,E2 33568.779} C_VEL
LIN {X 0,Y 703.906,Z 1048.264,A -85,B 0,C 180,E1 33567.069,E2 33567.069} C_VEL
LIN {X 0,Y 703.911,Z 1046.58,A -85,B 0,C 180,E1 33564.947,E2 33564.947} C_VEL
LIN {X 0,Y 703.91,Z 1043.716,A -85,B 0,C 180,E1 33563.179,E2 33563.179} C_VEL
LIN {X 0,Y 703.925,Z 1039.223,A -85,B 0,C 180,E1 33561.258,E2 33561.258} C_VEL
LIN {X 0,Y 703.944,Z 1033.051,A -85,B 0,C 180,E1 33559.359,E2 33559.359} C_VEL
LIN {X 0,Y 704.021,Z 1026.412,A -85,B 0,C 180,E1 33557.7,E2 33557.7} C_VEL
LIN {X 0,Y 704.132,Z 1016.7,A -85,B 0,C 180,E1 33555.695,E2 33555.695} C_VEL
LIN {X 0,Y 704.274,Z 1006.757,A -85,B 0,C 180,E1 33553.982,E2 33553.982} C_VEL
LIN {X 0,Y 704.507,Z 994.482,A -85,B 0,C 180,E1 33552.148,E2 33552.148} C_VEL
LIN {X 0,Y 704.771,Z 981.118,A -85,B 0,C 180,E1 33550.438,E2 33550.438} C_VEL
LIN {X 0,Y 705.153,Z 965.849,A -85,B 0,C 180,E1 33548.715,E2 33548.715} C_VEL
LIN {X 0,Y 705.59,Z 949.887,A -85,B 0,C 180,E1 33547.152,E2 33547.152} C_VEL
LIN {X 0,Y 706.101,Z 932.311,A -85,B 0,C 180,E1 33545.62,E2 33545.62} C_VEL
LIN {X 0,Y 706.671,Z 913.726,A -85,B 0,C 180,E1 33544.209,E2 33544.209} C_VEL
LIN {X 0,Y 707.3,Z 893.136,A -85,B 0,C 180,E1 33542.831,E2 33542.831} C_VEL
LIN {X 0,Y 707.937,Z 873.068,A -85,B 0,C 180,E1 33541.669,E2 33541.669} C_VEL
LIN {X 0,Y 708.616,Z 850.437,A -85,B 0,C 180,E1 33540.531,E2 33540.531} C_VEL
LIN {X 0,Y 709.191,Z 829.539,A -85,B 0,C 180,E1 33539.64,E2 33539.64} C_VEL
LIN {X 0,Y 709.837,Z 806.353,A -85,B 0,C 180,E1 33538.8,E2 33538.8} C_VEL
LIN {X 0,Y 710.287,Z 782.585,A -85,B 0,C 180,E1 33538.111,E2 33538.111} C_VEL
LIN {X 0,Y 710.813,Z 758.633,A -85,B 0,C 180,E1 33537.563,E2 33537.563} C_VEL
LIN {X 0,Y 711.111,Z 734.559,A -85,B 0,C 180,E1 33537.174,E2 33537.174} C_VEL
LIN {X 0,Y 712.578,Z 476.432,A -85,B 0,C 180,E1 33534.211,E2 33534.211} C_VEL
LIN {X 0,Y 713.043,Z 359.592,A -85,B 0,C 180,E1 33532.839,E2 33532.839} C_VEL
LIN {X 0,Y 709.987,Z 349.207,A -85,B 0,C 180,E1 33532.539,E2 33532.539} C_VEL
LIN {X 0,Y 709.008,Z 347.055,A -85,B 0,C 180,E1 33532.427,E2 33532.427} C_VEL
LIN {X 0,Y 704.303,Z 333.503,A -85,B 0,C 180,E1 33531.057,E2 33531.057} C_VEL
LIN {X 0,Y 704.295,Z 333.498,A -85,B 0,C 180,E1 33527.925,E2 33527.925} C_VEL
LIN {X 0,Y 704.277,Z 333.497,A -85,B 0,C 180,E1 33525.34,E2 33525.34} C_VEL
LIN {X 0,Y 704.344,Z 333.496,A -85,B 0,C 180,E1 33522.511,E2 33522.511} C_VEL
LIN {X 0,Y 704.281,Z 333.492,A -85,B 0,C 180,E1 33519.603,E2 33519.603} C_VEL
LIN {X 0,Y 704.286,Z 333.498,A -85,B 0,C 180,E1 33517.011,E2 33517.011} C_VEL
LIN {X 0,Y 704.331,Z 333.493,A -85,B 0,C 180,E1 33513.997,E2 33513.997} C_VEL
LIN {X 0,Y 704.274,Z 333.493,A -85,B 0,C 180,E1 33511.212,E2 33511.212} C_VEL
LIN {X 0,Y 704.324,Z 333.498,A -85,B 0,C 180,E1 33508.49,E2 33508.49} C_VEL
LIN {X 0,Y 704.284,Z 333.492,A -85,B 0,C 180,E1 33505.452,E2 33505.452} C_VEL
LIN {X 0,Y 704.279,Z 333.498,A -85,B 0,C 180,E1 33502.867,E2 33502.867} C_VEL
LIN {X 0,Y 704.345,Z 333.493,A -85,B 0,C 180,E1 33499.92,E2 33499.92} C_VEL
LIN {X 0,Y 704.274,Z 333.494,A -85,B 0,C 180,E1 33497.091,E2 33497.091} C_VEL
LIN {X 0,Y 704.296,Z 333.498,A -85,B 0,C 180,E1 33494.47,E2 33494.47} C_VEL
LIN {X 0,Y 704.301,Z 333.493,A -85,B 0,C 180,E1 33491.381,E2 33491.381} C_VEL
LIN {X 0,Y 704.274,Z 333.495,A -85,B 0,C 180,E1 33488.738,E2 33488.738} C_VEL
LIN {X 0,Y 704.342,Z 333.494,A -85,B 0,C 180,E1 33485.948,E2 33485.948} C_VEL
LIN {X 0,Y 704.28,Z 333.495,A -85,B 0,C 180,E1 33483.011,E2 33483.011} C_VEL
LIN {X 0,Y 704.281,Z 333.495,A -85,B 0,C 180,E1 33480.407,E2 33480.407} C_VEL
LIN {X 0,Y 704.337,Z 333.489,A -85,B 0,C 180,E1 33477.478,E2 33477.478} C_VEL
LIN {X 0,Y 704.273,Z 333.496,A -85,B 0,C 180,E1 33474.705,E2 33474.705} C_VEL
LIN {X 0,Y 704.295,Z 333.494,A -85,B 0,C 180,E1 33472.085,E2 33472.085} C_VEL
LIN {X 0,Y 704.293,Z 333.489,A -85,B 0,C 180,E1 33468.95,E2 33468.95} C_VEL
LIN {X 0,Y 704.272,Z 333.497,A -85,B 0,C 180,E1 33466.368,E2 33466.368} C_VEL
LIN {X 0,Y 704.34,Z 333.495,A -85,B 0,C 180,E1 33463.59,E2 33463.59} C_VEL
LIN {X 0,Y 704.28,Z 333.49,A -85,B 0,C 180,E1 33460.683,E2 33460.683} C_VEL
LIN {X 0,Y 704.277,Z 333.498,A -85,B 0,C 180,E1 33458.075,E2 33458.075} C_VEL
LIN {X 0,Y 704.343,Z 333.494,A -85,B 0,C 180,E1 33455.152,E2 33455.152} C_VEL
LIN {X 0,Y 704.273,Z 333.494,A -85,B 0,C 180,E1 33452.338,E2 33452.338} C_VEL
LIN {X 0,Y 704.292,Z 333.498,A -85,B 0,C 180,E1 33449.735,E2 33449.735} C_VEL
LIN {X 0,Y 704.293,Z 333.495,A -85,B 0,C 180,E1 33446.575,E2 33446.575} C_VEL
LIN {X 0,Y 704.271,Z 333.498,A -85,B 0,C 180,E1 33444,E2 33444} C_VEL
LIN {X 0,Y 704.346,Z 333.498,A -85,B 0,C 180,E1 33441.137,E2 33441.137} C_VEL
LIN {X 0,Y 704.278,Z 333.496,A -85,B 0,C 180,E1 33438.252,E2 33438.252} C_VEL
LIN {X 0,Y 704.278,Z 333.499,A -85,B 0,C 180,E1 33435.688,E2 33435.688} C_VEL
LIN {X 0,Y 704.338,Z 333.493,A -85,B 0,C 180,E1 33432.733,E2 33432.733} C_VEL
LIN {X 0,Y 704.272,Z 333.502,A -85,B 0,C 180,E1 33429.921,E2 33429.921} C_VEL
LIN {X 0,Y 704.343,Z 333.517,A -85,B 0,C 180,E1 33429.007,E2 33429.007} C_VEL
LIN {X 0,Y 710.717,Z 350.76,A -85,B 0,C 180,E1 33427.327,E2 33427.327} C_VEL
LIN {X 0,Y 710.234,Z 377.393,A -85,B 0,C 180,E1 33425.424,E2 33425.424} C_VEL
LIN {X 0,Y 713.272,Z 390.551,A -85,B 0,C 180,E1 33425.091,E2 33425.091} C_VEL
LIN {X 0,Y 711.768,Z 650.758,A -85,B 0,C 180,E1 33422.087,E2 33422.087} C_VEL
LIN {X 0,Y 711.095,Z 767.217,A -85,B 0,C 180,E1 33420.746,E2 33420.746} C_VEL
LIN {X 0,Y 710.679,Z 792.763,A -85,B 0,C 180,E1 33420.306,E2 33420.306} C_VEL
LIN {X 0,Y 710.262,Z 814.452,A -85,B 0,C 180,E1 33419.795,E2 33419.795} C_VEL
LIN {X 0,Y 709.764,Z 838.564,A -85,B 0,C 180,E1 33419.08,E2 33419.08} C_VEL
LIN {X 0,Y 709.16,Z 860.49,A -85,B 0,C 180,E1 33418.278,E2 33418.278} C_VEL
LIN {X 0,Y 708.561,Z 883.171,A -85,B 0,C 180,E1 33417.298,E2 33417.298} C_VEL
LIN {X 0,Y 707.876,Z 904.76,A -85,B 0,C 180,E1 33416.194,E2 33416.194} C_VEL
LIN {X 0,Y 707.237,Z 925.752,A -85,B 0,C 180,E1 33414.962,E2 33414.962} C_VEL
LIN {X 0,Y 706.621,Z 945.052,A -85,B 0,C 180,E1 33413.651,E2 33413.651} C_VEL
LIN {X 0,Y 706.067,Z 963.763,A -85,B 0,C 180,E1 33412.217,E2 33412.217} C_VEL
LIN {X 0,Y 705.557,Z 980.805,A -85,B 0,C 180,E1 33410.718,E2 33410.718} C_VEL
LIN {X 0,Y 705.128,Z 996.967,A -85,B 0,C 180,E1 33409.121,E2 33409.121} C_VEL
LIN {X 0,Y 704.773,Z 1011.224,A -85,B 0,C 180,E1 33407.504,E2 33407.504} C_VEL
LIN {X 0,Y 704.503,Z 1025.061,A -85,B 0,C 180,E1 33405.729,E2 33405.729} C_VEL
LIN {X 0,Y 704.267,Z 1036.798,A -85,B 0,C 180,E1 33403.967,E2 33403.967} C_VEL
LIN {X 0,Y 704.122,Z 1046.947,A -85,B 0,C 180,E1 33402.215,E2 33402.215} C_VEL
LIN {X 0,Y 704.017,Z 1056.539,A -85,B 0,C 180,E1 33400.226,E2 33400.226} C_VEL
LIN {X 0,Y 703.947,Z 1063.12,A -85,B 0,C 180,E1 33398.577,E2 33398.577} C_VEL
LIN {X 0,Y 703.913,Z 1069.451,A -85,B 0,C 180,E1 33396.607,E2 33396.607} C_VEL
LIN {X 0,Y 703.919,Z 1073.814,A -85,B 0,C 180,E1 33394.726,E2 33394.726} C_VEL
LIN {X 0,Y 703.909,Z 1076.797,A -85,B 0,C 180,E1 33392.85,E2 33392.85} C_VEL
LIN {X 0,Y 703.902,Z 1078.284,A -85,B 0,C 180,E1 33390.814,E2 33390.814} C_VEL
LIN {X 0,Y 703.907,Z 1078.262,A -85,B 0,C 180,E1 33389.105,E2 33389.105} C_VEL
LIN {X 0,Y 703.916,Z 1076.573,A -85,B 0,C 180,E1 33386.987,E2 33386.987} C_VEL
LIN {X 0,Y 703.919,Z 1073.655,A -85,B 0,C 180,E1 33385.193,E2 33385.193} C_VEL
LIN {X 0,Y 703.921,Z 1069.015,A -85,B 0,C 180,E1 33383.229,E2 33383.229} C_VEL
LIN {X 0,Y 703.945,Z 1062.815,A -85,B 0,C 180,E1 33381.34,E2 33381.34} C_VEL
LIN {X 0,Y 704.025,Z 1056.183,A -85,B 0,C 180,E1 33379.691,E2 33379.691} C_VEL
LIN {X 0,Y 704.13,Z 1046.399,A -85,B 0,C 180,E1 33377.685,E2 33377.685} C_VEL
LIN {X 0,Y 704.267,Z 1036.8,A -85,B 0,C 180,E1 33376.033,E2 33376.033} C_VEL
LIN {X 0,Y 704.511,Z 1024.439,A -85,B 0,C 180,E1 33374.187,E2 33374.187} C_VEL
LIN {X 0,Y 704.773,Z 1011.224,A -85,B 0,C 180,E1 33372.496,E2 33372.496} C_VEL
LIN {X 0,Y 705.147,Z 996.175,A -85,B 0,C 180,E1 33370.794,E2 33370.794} C_VEL
LIN {X 0,Y 705.592,Z 979.534,A -85,B 0,C 180,E1 33369.164,E2 33369.164} C_VEL
LIN {X 0,Y 706.116,Z 961.607,A -85,B 0,C 180,E1 33367.61,E2 33367.61} C_VEL
LIN {X 0,Y 706.659,Z 944.007,A -85,B 0,C 180,E1 33366.274,E2 33366.274} C_VEL
LIN {X 0,Y 707.287,Z 923.622,A -85,B 0,C 180,E1 33364.906,E2 33364.906} C_VEL
LIN {X 0,Y 707.908,Z 903.833,A -85,B 0,C 180,E1 33363.756,E2 33363.756} C_VEL
LIN {X 0,Y 708.586,Z 882.24,A -85,B 0,C 180,E1 33362.657,E2 33362.657} C_VEL
LIN {X 0,Y 709.159,Z 860.493,A -85,B 0,C 180,E1 33361.722,E2 33361.722} C_VEL
LIN {X 0,Y 709.764,Z 838.565,A -85,B 0,C 180,E1 33360.92,E2 33360.92} C_VEL
LIN {X 0,Y 710.264,Z 814.228,A -85,B 0,C 180,E1 33360.199,E2 33360.199} C_VEL
LIN {X 0,Y 710.693,Z 792.376,A -85,B 0,C 180,E1 33359.686,E2 33359.686} C_VEL
LIN {X 0,Y 711.097,Z 767.07,A -85,B 0,C 180,E1 33359.252,E2 33359.252} C_VEL
LIN {X 0,Y 711.941,Z 619.333,A -85,B 0,C 180,E1 33357.554,E2 33357.554} C_VEL
LIN {X 0,Y 713.239,Z 389.492,A -85,B 0,C 180,E1 33354.894,E2 33354.894} C_VEL
LIN {X 0,Y 710.16,Z 376.685,A -85,B 0,C 180,E1 33354.543,E2 33354.543} C_VEL
LIN {X 0,Y 710.659,Z 350.511,A -85,B 0,C 180,E1 33352.651,E2 33352.651} C_VEL
LIN {X 0,Y 704.337,Z 333.5,A -85,B 0,C 180,E1 33350.961,E2 33350.961} C_VEL
LIN {X 0,Y 704.27,Z 333.501,A -85,B 0,C 180,E1 33348.142,E2 33348.142} C_VEL
LIN {X 0,Y 704.314,Z 333.497,A -85,B 0,C 180,E1 33345.453,E2 33345.453} C_VEL
LIN {X 0,Y 704.286,Z 333.5,A -85,B 0,C 180,E1 33342.405,E2 33342.405} C_VEL
LIN {X 0,Y 704.272,Z 333.494,A -85,B 0,C 180,E1 33339.815,E2 33339.815} C_VEL
LIN {X 0,Y 704.345,Z 333.493,A -85,B 0,C 180,E1 33336.943,E2 33336.943} C_VEL
LIN {X 0,Y 704.276,Z 333.496,A -85,B 0,C 180,E1 33334.111,E2 33334.111} C_VEL
LIN {X 0,Y 704.281,Z 333.494,A -85,B 0,C 180,E1 33331.498,E2 33331.498} C_VEL
LIN {X 0,Y 704.326,Z 333.496,A -85,B 0,C 180,E1 33328.49,E2 33328.49} C_VEL
LIN {X 0,Y 704.271,Z 333.496,A -85,B 0,C 180,E1 33325.75,E2 33325.75} C_VEL
LIN {X 0,Y 704.329,Z 333.488,A -85,B 0,C 180,E1 33322.98,E2 33322.98} C_VEL
LIN {X 0,Y 704.283,Z 333.494,A -85,B 0,C 180,E1 33319.972,E2 33319.972} C_VEL
LIN {X 0,Y 704.279,Z 333.495,A -85,B 0,C 180,E1 33317.346,E2 33317.346} C_VEL
LIN {X 0,Y 704.343,Z 333.493,A -85,B 0,C 180,E1 33314.385,E2 33314.385} C_VEL
LIN {X 0,Y 704.273,Z 333.496,A -85,B 0,C 180,E1 33311.548,E2 33311.548} C_VEL
LIN {X 0,Y 704.316,Z 333.487,A -85,B 0,C 180,E1 33308.82,E2 33308.82} C_VEL
LIN {X 0,Y 704.288,Z 333.495,A -85,B 0,C 180,E1 33305.785,E2 33305.785} C_VEL
LIN {X 0,Y 704.276,Z 333.493,A -85,B 0,C 180,E1 33303.174,E2 33303.174} C_VEL
LIN {X 0,Y 704.347,Z 333.496,A -85,B 0,C 180,E1 33300.244,E2 33300.244} C_VEL
LIN {X 0,Y 704.275,Z 333.497,A -85,B 0,C 180,E1 33297.396,E2 33297.396} C_VEL
LIN {X 0,Y 704.293,Z 333.491,A -85,B 0,C 180,E1 33294.787,E2 33294.787} C_VEL
LIN {X 0,Y 704.302,Z 333.499,A -85,B 0,C 180,E1 33291.674,E2 33291.674} C_VEL
LIN {X 0,Y 704.273,Z 333.489,A -85,B 0,C 180,E1 33289.033,E2 33289.033} C_VEL
LIN {X 0,Y 704.344,Z 333.493,A -85,B 0,C 180,E1 33286.17,E2 33286.17} C_VEL
LIN {X 0,Y 704.279,Z 333.495,A -85,B 0,C 180,E1 33283.249,E2 33283.249} C_VEL
LIN {X 0,Y 704.29,Z 333.494,A -85,B 0,C 180,E1 33280.597,E2 33280.597} C_VEL
LIN {X 0,Y 704.336,Z 333.488,A -85,B 0,C 180,E1 33278.153,E2 33278.153} C_VEL
LIN {X 0,Y 703.381,Z 333.617,A -85,B 0,C 180,E1 33277.527,E2 33277.527} C_VEL
LIN {X 0,Y 696.926,Z 334.421,A -85,B 0,C 180,E1 33275.772,E2 33275.772} C_VEL
LIN {X 0,Y 696.356,Z 334.481,A -85,B 0,C 180,E1 33275.316,E2 33275.316} C_VEL
LIN {X 0,Y 696.341,Z 334.484,A -85,B 0,C 180,E1 33272.645,E2 33272.645} C_VEL
LIN {X 0,Y 696.407,Z 334.479,A -85,B 0,C 180,E1 33269.737,E2 33269.737} C_VEL
LIN {X 0,Y 696.337,Z 334.481,A -85,B 0,C 180,E1 33266.832,E2 33266.832} C_VEL
LIN {X 0,Y 696.384,Z 334.482,A -85,B 0,C 180,E1 33264.037,E2 33264.037} C_VEL
LIN {X 0,Y 696.349,Z 334.486,A -85,B 0,C 180,E1 33260.971,E2 33260.971} C_VEL
LIN {X 0,Y 696.346,Z 334.486,A -85,B 0,C 180,E1 33258.303,E2 33258.303} C_VEL
LIN {X 0,Y 696.393,Z 334.471,A -85,B 0,C 180,E1 33255.287,E2 33255.287} C_VEL
LIN {X 0,Y 696.339,Z 334.485,A -85,B 0,C 180,E1 33252.555,E2 33252.555} C_VEL
LIN {X 0,Y 696.384,Z 334.485,A -85,B 0,C 180,E1 33249.81,E2 33249.81} C_VEL
LIN {X 0,Y 696.353,Z 334.493,A -85,B 0,C 180,E1 33246.752,E2 33246.752} C_VEL
LIN {X 0,Y 696.422,Z 334.619,A -85,B 0,C 180,E1 33245.252,E2 33245.252} C_VEL
LIN {X 0,Y 701.138,Z 347.973,A -85,B 0,C 180,E1 33243.902,E2 33243.902} C_VEL
LIN {X 0,Y 704.636,Z 354.675,A -85,B 0,C 180,E1 33243.614,E2 33243.614} C_VEL
LIN {X 0,Y 706.663,Z 363.004,A -85,B 0,C 180,E1 33243.394,E2 33243.394} C_VEL
LIN {X 0,Y 705.128,Z 598.248,A -85,B 0,C 180,E1 33240.648,E2 33240.648} C_VEL
LIN {X 0,Y 704.21,Z 737.177,A -85,B 0,C 180,E1 33239.035,E2 33239.035} C_VEL
LIN {X 0,Y 703.751,Z 762.768,A -85,B 0,C 180,E1 33238.591,E2 33238.591} C_VEL
LIN {X 0,Y 703.256,Z 784.577,A -85,B 0,C 180,E1 33238.074,E2 33238.074} C_VEL
LIN {X 0,Y 702.693,Z 808.39,A -85,B 0,C 180,E1 33237.362,E2 33237.362} C_VEL
LIN {X 0,Y 702.015,Z 830.201,A -85,B 0,C 180,E1 33236.559,E2 33236.559} C_VEL
LIN {X 0,Y 701.319,Z 852.473,A -85,B 0,C 180,E1 33235.594,E2 33235.594} C_VEL
LIN {X 0,Y 700.562,Z 873.84,A -85,B 0,C 180,E1 33234.495,E2 33234.495} C_VEL
LIN {X 0,Y 699.805,Z 894.874,A -85,B 0,C 180,E1 33233.259,E2 33233.259} C_VEL
LIN {X 0,Y 699.102,Z 914.473,A -85,B 0,C 180,E1 33231.919,E2 33231.919} C_VEL
LIN {X 0,Y 698.425,Z 933.56,A -85,B 0,C 180,E1 33230.446,E2 33230.446} C_VEL
LIN {X 0,Y 697.838,Z 951.002,A -85,B 0,C 180,E1 33228.894,E2 33228.894} C_VEL
LIN {X 0,Y 697.32,Z 967.342,A -85,B 0,C 180,E1 33227.257,E2 33227.257} C_VEL
LIN {X 0,Y 696.899,Z 982.046,A -85,B 0,C 180,E1 33225.563,E2 33225.563} C_VEL
LIN {X 0,Y 696.566,Z 996.198,A -85,B 0,C 180,E1 33223.701,E2 33223.701} C_VEL
LIN {X 0,Y 696.32,Z 1007.726,A -85,B 0,C 180,E1 33221.934,E2 33221.934} C_VEL
LIN {X 0,Y 696.141,Z 1018.549,A -85,B 0,C 180,E1 33220.009,E2 33220.009} C_VEL
LIN {X 0,Y 696.031,Z 1027.063,A -85,B 0,C 180,E1 33218.176,E2 33218.176} C_VEL
LIN {X 0,Y 695.956,Z 1033.838,A -85,B 0,C 180,E1 33216.434,E2 33216.434} C_VEL
LIN {X 0,Y 695.923,Z 1040.196,A -85,B 0,C 180,E1 33214.339,E2 33214.339} C_VEL
LIN {X 0,Y 695.916,Z 1044.164,A -85,B 0,C 180,E1 33212.553,E2 33212.553} C_VEL
LIN {X 0,Y 695.896,Z 1047.103,A -85,B 0,C 180,E1 33210.576,E2 33210.576} C_VEL
LIN {X 0,Y 695.895,Z 1048.31,A -85,B 0,C 180,E1 33208.683,E2 33208.683} C_VEL
LIN {X 0,Y 695.91,Z 1048.212,A -85,B 0,C 180,E1 33206.87,E2 33206.87} C_VEL
LIN {X 0,Y 695.91,Z 1046.435,A -85,B 0,C 180,E1 33204.807,E2 33204.807} C_VEL
LIN {X 0,Y 695.91,Z 1043.609,A -85,B 0,C 180,E1 33203.068,E2 33203.068} C_VEL
LIN {X 0,Y 695.938,Z 1038.914,A -85,B 0,C 180,E1 33201.073,E2 33201.073} C_VEL
LIN {X 0,Y 695.953,Z 1032.963,A -85,B 0,C 180,E1 33199.235,E2 33199.235} C_VEL
LIN {X 0,Y 696.045,Z 1026.31,A -85,B 0,C 180,E1 33197.556,E2 33197.556} C_VEL
LIN {X 0,Y 696.178,Z 1016.28,A -85,B 0,C 180,E1 33195.476,E2 33195.476} C_VEL
LIN {X 0,Y 696.349,Z 1006.27,A -85,B 0,C 180,E1 33193.74,E2 33193.74} C_VEL
LIN {X 0,Y 696.617,Z 993.585,A -85,B 0,C 180,E1 33191.843,E2 33191.843} C_VEL
LIN {X 0,Y 696.966,Z 980.195,A -85,B 0,C 180,E1 33190.123,E2 33190.123} C_VEL
LIN {X 0,Y 697.425,Z 963.824,A -85,B 0,C 180,E1 33188.285,E2 33188.285} C_VEL
LIN {X 0,Y 697.931,Z 948.197,A -85,B 0,C 180,E1 33186.753,E2 33186.753} C_VEL
LIN {X 0,Y 698.567,Z 929.18,A -85,B 0,C 180,E1 33185.114,E2 33185.114} C_VEL
LIN {X 0,Y 699.202,Z 911.507,A -85,B 0,C 180,E1 33183.776,E2 33183.776} C_VEL
LIN {X 0,Y 699.962,Z 890.491,A -85,B 0,C 180,E1 33182.384,E2 33182.384} C_VEL
LIN {X 0,Y 700.64,Z 871.756,A -85,B 0,C 180,E1 33181.3,E2 33181.3} C_VEL
LIN {X 0,Y 701.397,Z 849.133,A -85,B 0,C 180,E1 33180.164,E2 33180.164} C_VEL
LIN {X 0,Y 702.059,Z 828.842,A -85,B 0,C 180,E1 33179.297,E2 33179.297} C_VEL
LIN {X 0,Y 702.771,Z 806.24,A -85,B 0,C 180,E1 33178.475,E2 33178.475} C_VEL
LIN {X 0,Y 703.296,Z 782.52,A -85,B 0,C 180,E1 33177.782,E2 33177.782} C_VEL
LIN {X 0,Y 703.893,Z 758.545,A -85,B 0,C 180,E1 33177.231,E2 33177.231} C_VEL
LIN {X 0,Y 704.229,Z 734.414,A -85,B 0,C 180,E1 33176.838,E2 33176.838} C_VEL
LIN {X 0,Y 705.908,Z 478.384,A -85,B 0,C 180,E1 33173.873,E2 33173.873} C_VEL
LIN {X 0,Y 706.499,Z 361.579,A -85,B 0,C 180,E1 33172.489,E2 33172.489} C_VEL
LIN {X 0,Y 703.911,Z 352.9,A -85,B 0,C 180,E1 33172.232,E2 33172.232} C_VEL
LIN {X 0,Y 700.814,Z 347.209,A -85,B 0,C 180,E1 33171.959,E2 33171.959} C_VEL
LIN {X 0,Y 696.408,Z 334.488,A -85,B 0,C 180,E1 33170.627,E2 33170.627} C_VEL
LIN {X 0,Y 696.341,Z 334.489,A -85,B 0,C 180,E1 33167.689,E2 33167.689} C_VEL
LIN {X 0,Y 696.354,Z 334.487,A -85,B 0,C 180,E1 33165.052,E2 33165.052} C_VEL
LIN {X 0,Y 696.367,Z 334.48,A -85,B 0,C 180,E1 33161.946,E2 33161.946} C_VEL
LIN {X 0,Y 696.336,Z 334.482,A -85,B 0,C 180,E1 33159.289,E2 33159.289} C_VEL
LIN {X 0,Y 696.398,Z 334.472,A -85,B 0,C 180,E1 33156.472,E2 33156.472} C_VEL
LIN {X 0,Y 696.347,Z 334.484,A -85,B 0,C 180,E1 33153.561,E2 33153.561} C_VEL
LIN {X 0,Y 696.344,Z 334.483,A -85,B 0,C 180,E1 33150.935,E2 33150.935} C_VEL
LIN {X 0,Y 696.408,Z 334.481,A -85,B 0,C 180,E1 33147.993,E2 33147.993} C_VEL
LIN {X 0,Y 696.335,Z 334.482,A -85,B 0,C 180,E1 33145.153,E2 33145.153} C_VEL
LIN {X 0,Y 696.389,Z 334.487,A -85,B 0,C 180,E1 33142.364,E2 33142.364} C_VEL
LIN {X 0,Y 696.349,Z 334.483,A -85,B 0,C 180,E1 33139.371,E2 33139.371} C_VEL
LIN {X 0,Y 696.342,Z 334.485,A -85,B 0,C 180,E1 33136.713,E2 33136.713} C_VEL
LIN {X 0,Y 696.396,Z 334.48,A -85,B 0,C 180,E1 33133.704,E2 33133.704} C_VEL
LIN {X 0,Y 696.334,Z 334.484,A -85,B 0,C 180,E1 33130.926,E2 33130.926} C_VEL
LIN {X 0,Y 696.381,Z 334.487,A -85,B 0,C 180,E1 33128.172,E2 33128.172} C_VEL
LIN {X 0,Y 696.345,Z 334.481,A -85,B 0,C 180,E1 33125.108,E2 33125.108} C_VEL
LIN {X 0,Y 696.341,Z 334.487,A -85,B 0,C 180,E1 33122.469,E2 33122.469} C_VEL
LIN {X 0,Y 696.404,Z 334.482,A -85,B 0,C 180,E1 33119.506,E2 33119.506} C_VEL
LIN {X 0,Y 696.333,Z 334.48,A -85,B 0,C 180,E1 33116.707,E2 33116.707} C_VEL
LIN {X 0,Y 696.373,Z 334.489,A -85,B 0,C 180,E1 33113.983,E2 33113.983} C_VEL
LIN {X 0,Y 696.348,Z 334.484,A -85,B 0,C 180,E1 33110.912,E2 33110.912} C_VEL
LIN {X 0,Y 696.335,Z 334.481,A -85,B 0,C 180,E1 33108.319,E2 33108.319} C_VEL
LIN {X 0,Y 696.406,Z 334.478,A -85,B 0,C 180,E1 33105.402,E2 33105.402} C_VEL
LIN {X 0,Y 696.335,Z 334.485,A -85,B 0,C 180,E1 33102.536,E2 33102.536} C_VEL
LIN {X 0,Y 696.354,Z 334.482,A -85,B 0,C 180,E1 33099.897,E2 33099.897} C_VEL
LIN {X 0,Y 696.353,Z 334.479,A -85,B 0,C 180,E1 33096.742,E2 33096.742} C_VEL
LIN {X 0,Y 696.335,Z 334.486,A -85,B 0,C 180,E1 33094.118,E2 33094.118} C_VEL
LIN {X 0,Y 696.409,Z 334.485,A -85,B 0,C 180,E1 33091.25,E2 33091.25} C_VEL
LIN {X 0,Y 696.335,Z 334.485,A -85,B 0,C 180,E1 33088.376,E2 33088.376} C_VEL
LIN {X 0,Y 696.346,Z 334.489,A -85,B 0,C 180,E1 33085.745,E2 33085.745} C_VEL
LIN {X 0,Y 696.377,Z 334.483,A -85,B 0,C 180,E1 33082.699,E2 33082.699} C_VEL
LIN {X 0,Y 696.333,Z 334.487,A -85,B 0,C 180,E1 33079.961,E2 33079.961} C_VEL
LIN {X 0,Y 696.399,Z 334.481,A -85,B 0,C 180,E1 33077.112,E2 33077.112} C_VEL
LIN {X 0,Y 696.337,Z 334.487,A -85,B 0,C 180,E1 33074.141,E2 33074.141} C_VEL
LIN {X 0,Y 696.342,Z 334.491,A -85,B 0,C 180,E1 33071.559,E2 33071.559} C_VEL
LIN {X 0,Y 696.357,Z 334.56,A -85,B 0,C 180,E1 33069.441,E2 33069.441} C_VEL
LIN {X 0,Y 703.699,Z 354.082,A -85,B 0,C 180,E1 33067.507,E2 33067.507} C_VEL
LIN {X 0,Y 703.258,Z 377.512,A -85,B 0,C 180,E1 33065.827,E2 33065.827} C_VEL
LIN {X 0,Y 706.709,Z 392.231,A -85,B 0,C 180,E1 33065.446,E2 33065.446} C_VEL
LIN {X 0,Y 704.974,Z 652.667,A -85,B 0,C 180,E1 33062.412,E2 33062.412} C_VEL
LIN {X 0,Y 704.209,Z 767.356,A -85,B 0,C 180,E1 33061.078,E2 33061.078} C_VEL
LIN {X 0,Y 703.745,Z 792.891,A -85,B 0,C 180,E1 33060.633,E2 33060.633} C_VEL
LIN {X 0,Y 703.253,Z 814.671,A -85,B 0,C 180,E1 33060.117,E2 33060.117} C_VEL
LIN {X 0,Y 702.689,Z 838.561,A -85,B 0,C 180,E1 33059.401,E2 33059.401} C_VEL
LIN {X 0,Y 702.044,Z 859.357,A -85,B 0,C 180,E1 33058.637,E2 33058.637} C_VEL
LIN {X 0,Y 701.345,Z 881.247,A -85,B 0,C 180,E1 33057.695,E2 33057.695} C_VEL
LIN {X 0,Y 700.588,Z 903.141,A -85,B 0,C 180,E1 33056.579,E2 33056.579} C_VEL
LIN {X 0,Y 699.874,Z 922.83,A -85,B 0,C 180,E1 33055.429,E2 33055.429} C_VEL
LIN {X 0,Y 699.142,Z 943.233,A -85,B 0,C 180,E1 33054.054,E2 33054.054} C_VEL
LIN {X 0,Y 698.498,Z 961.254,A -85,B 0,C 180,E1 33052.676,E2 33052.676} C_VEL
LIN {X 0,Y 697.901,Z 978.856,A -85,B 0,C 180,E1 33051.14,E2 33051.14} C_VEL
LIN {X 0,Y 697.402,Z 994.485,A -85,B 0,C 180,E1 33049.603,E2 33049.603} C_VEL
LIN {X 0,Y 696.975,Z 1009.811,A -85,B 0,C 180,E1 33047.879,E2 33047.879} C_VEL
LIN {X 0,Y 696.626,Z 1022.853,A -85,B 0,C 180,E1 33046.21,E2 33046.21} C_VEL
LIN {X 0,Y 696.344,Z 1036.08,A -85,B 0,C 180,E1 33044.246,E2 33044.246} C_VEL
LIN {X 0,Y 696.176,Z 1046.028,A -85,B 0,C 180,E1 33042.526,E2 33042.526} C_VEL
LIN {X 0,Y 696.049,Z 1055.829,A -85,B 0,C 180,E1 33040.512,E2 33040.512} C_VEL
LIN {X 0,Y 695.954,Z 1062.816,A -85,B 0,C 180,E1 33038.76,E2 33038.76} C_VEL
LIN {X 0,Y 695.931,Z 1069.015,A -85,B 0,C 180,E1 33036.849,E2 33036.849} C_VEL
LIN {X 0,Y 695.92,Z 1073.656,A -85,B 0,C 180,E1 33034.863,E2 33034.863} C_VEL
LIN {X 0,Y 695.916,Z 1076.573,A -85,B 0,C 180,E1 33033.047,E2 33033.047} C_VEL
LIN {X 0,Y 695.907,Z 1078.262,A -85,B 0,C 180,E1 33030.906,E2 33030.906} C_VEL
LIN {X 0,Y 695.902,Z 1078.284,A -85,B 0,C 180,E1 33029.177,E2 33029.177} C_VEL
LIN {X 0,Y 695.91,Z 1076.797,A -85,B 0,C 180,E1 33027.117,E2 33027.117} C_VEL
LIN {X 0,Y 695.92,Z 1073.814,A -85,B 0,C 180,E1 33025.22,E2 33025.22} C_VEL
LIN {X 0,Y 695.918,Z 1069.451,A -85,B 0,C 180,E1 33023.317,E2 33023.317} C_VEL
LIN {X 0,Y 695.953,Z 1063.12,A -85,B 0,C 180,E1 33021.324,E2 33021.324} C_VEL
LIN {X 0,Y 696.042,Z 1056.539,A -85,B 0,C 180,E1 33019.655,E2 33019.655} C_VEL
LIN {X 0,Y 696.163,Z 1046.947,A -85,B 0,C 180,E1 33017.643,E2 33017.643} C_VEL
LIN {X 0,Y 696.329,Z 1036.802,A -85,B 0,C 180,E1 33015.871,E2 33015.871} C_VEL
LIN {X 0,Y 696.605,Z 1024.438,A -85,B 0,C 180,E1 33014.003,E2 33014.003} C_VEL
LIN {X 0,Y 696.931,Z 1011.226,A -85,B 0,C 180,E1 33012.293,E2 33012.293} C_VEL
LIN {X 0,Y 697.354,Z 996.174,A -85,B 0,C 180,E1 33010.57,E2 33010.57} C_VEL
LIN {X 0,Y 697.847,Z 980.463,A -85,B 0,C 180,E1 33009.01,E2 33009.01} C_VEL
LIN {X 0,Y 698.456,Z 962.713,A -85,B 0,C 180,E1 33007.439,E2 33007.439} C_VEL
LIN {X 0,Y 699.099,Z 944.448,A -85,B 0,C 180,E1 33006.034,E2 33006.034} C_VEL
LIN {X 0,Y 699.821,Z 924.352,A -85,B 0,C 180,E1 33004.664,E2 33004.664} C_VEL
LIN {X 0,Y 700.556,Z 903.948,A -85,B 0,C 180,E1 33003.465,E2 33003.465} C_VEL
LIN {X 0,Y 701.324,Z 882.242,A -85,B 0,C 180,E1 33002.35,E2 33002.35} C_VEL
LIN {X 0,Y 702.005,Z 860.492,A -85,B 0,C 180,E1 33001.408,E2 33001.408} C_VEL
LIN {X 0,Y 702.641,Z 839.846,A -85,B 0,C 180,E1 33000.644,E2 33000.644} C_VEL
LIN {X 0,Y 703.252,Z 814.781,A -85,B 0,C 180,E1 32999.886,E2 32999.886} C_VEL
LIN {X 0,Y 703.742,Z 793.026,A -85,B 0,C 180,E1 32999.37,E2 32999.37} C_VEL
LIN {X 0,Y 704.209,Z 767.542,A -85,B 0,C 180,E1 32998.925,E2 32998.925} C_VEL
LIN {X 0,Y 704.904,Z 663.834,A -85,B 0,C 180,E1 32997.717,E2 32997.717} C_VEL
LIN {X 0,Y 706.665,Z 398.597,A -85,B 0,C 180,E1 32994.63,E2 32994.63} C_VEL
LIN {X 0,Y 706.506,Z 390.587,A -85,B 0,C 180,E1 32994.523,E2 32994.523} C_VEL
LIN {X 0,Y 703.158,Z 376.685,A -85,B 0,C 180,E1 32994.136,E2 32994.136} C_VEL
LIN {X 0,Y 703.622,Z 353.739,A -85,B 0,C 180,E1 32992.463,E2 32992.463} C_VEL
LIN {X 0,Y 696.347,Z 334.498,A -85,B 0,C 180,E1 32990.538,E2 32990.538} C_VEL
LIN {X 0,Y 696.335,Z 334.49,A -85,B 0,C 180,E1 32987.935,E2 32987.935} C_VEL
LIN {X 0,Y 696.408,Z 334.488,A -85,B 0,C 180,E1 32985.057,E2 32985.057} C_VEL
LIN {X 0,Y 696.335,Z 334.489,A -85,B 0,C 180,E1 32982.188,E2 32982.188} C_VEL
LIN {X 0,Y 696.351,Z 334.481,A -85,B 0,C 180,E1 32979.549,E2 32979.549} C_VEL
LIN {X 0,Y 696.355,Z 334.489,A -85,B 0,C 180,E1 32976.372,E2 32976.372} C_VEL
LIN {X 0,Y 696.334,Z 334.483,A -85,B 0,C 180,E1 32973.757,E2 32973.757} C_VEL
LIN {X 0,Y 696.406,Z 334.481,A -85,B 0,C 180,E1 32970.932,E2 32970.932} C_VEL
LIN {X 0,Y 696.336,Z 334.482,A -85,B 0,C 180,E1 32967.982,E2 32967.982} C_VEL
LIN {X 0,Y 696.351,Z 334.483,A -85,B 0,C 180,E1 32965.334,E2 32965.334} C_VEL
LIN {X 0,Y 696.36,Z 334.488,A -85,B 0,C 180,E1 32962.188,E2 32962.188} C_VEL
LIN {X 0,Y 696.332,Z 334.481,A -85,B 0,C 180,E1 32959.547,E2 32959.547} C_VEL
LIN {X 0,Y 696.404,Z 334.483,A -85,B 0,C 180,E1 32956.688,E2 32956.688} C_VEL
LIN {X 0,Y 696.339,Z 334.484,A -85,B 0,C 180,E1 32953.79,E2 32953.79} C_VEL
LIN {X 0,Y 696.344,Z 334.484,A -85,B 0,C 180,E1 32951.178,E2 32951.178} C_VEL
LIN {X 0,Y 696.391,Z 334.487,A -85,B 0,C 180,E1 32948.172,E2 32948.172} C_VEL
LIN {X 0,Y 696.335,Z 334.482,A -85,B 0,C 180,E1 32945.438,E2 32945.438} C_VEL
LIN {X 0,Y 696.387,Z 334.48,A -85,B 0,C 180,E1 32942.633,E2 32942.633} C_VEL
LIN {X 0,Y 696.35,Z 334.479,A -85,B 0,C 180,E1 32939.671,E2 32939.671} C_VEL
LIN {X 0,Y 696.339,Z 334.484,A -85,B 0,C 180,E1 32937.037,E2 32937.037} C_VEL
LIN {X 0,Y 696.404,Z 334.48,A -85,B 0,C 180,E1 32934.066,E2 32934.066} C_VEL
LIN {X 0,Y 696.335,Z 334.486,A -85,B 0,C 180,E1 32931.245,E2 32931.245} C_VEL
LIN {X 0,Y 696.377,Z 334.474,A -85,B 0,C 180,E1 32928.487,E2 32928.487} C_VEL
LIN {X 0,Y 696.35,Z 334.485,A -85,B 0,C 180,E1 32925.42,E2 32925.42} C_VEL
LIN {X 0,Y 696.341,Z 334.482,A -85,B 0,C 180,E1 32922.794,E2 32922.794} C_VEL
LIN {X 0,Y 696.407,Z 334.483,A -85,B 0,C 180,E1 32919.843,E2 32919.843} C_VEL
LIN {X 0,Y 696.337,Z 334.486,A -85,B 0,C 180,E1 32916.989,E2 32916.989} C_VEL
LIN {X 0,Y 696.356,Z 334.481,A -85,B 0,C 180,E1 32915.316,E2 32915.316} C_VEL
LIN {X 0,Y 695.32,Z 334.607,A -85,B 0,C 180,E1 32914.682,E2 32914.682} C_VEL
LIN {X 0,Y 688.91,Z 335.413,A -85,B 0,C 180,E1 32912.905,E2 32912.905} C_VEL
LIN {X 0,Y 688.415,Z 335.473,A -85,B 0,C 180,E1 32912.444,E2 32912.444} C_VEL
LIN {X 0,Y 688.427,Z 335.478,A -85,B 0,C 180,E1 32909.298,E2 32909.298} C_VEL
LIN {X 0,Y 688.4,Z 335.468,A -85,B 0,C 180,E1 32906.599,E2 32906.599} C_VEL
LIN {X 0,Y 688.466,Z 335.473,A -85,B 0,C 180,E1 32903.661,E2 32903.661} C_VEL
LIN {X 0,Y 688.401,Z 335.473,A -85,B 0,C 180,E1 32900.73,E2 32900.73} C_VEL
LIN {X 0,Y 688.441,Z 335.473,A -85,B 0,C 180,E1 32897.967,E2 32897.967} C_VEL
LIN {X 0,Y 688.414,Z 335.469,A -85,B 0,C 180,E1 32894.902,E2 32894.902} C_VEL
LIN {X 0,Y 688.408,Z 335.472,A -85,B 0,C 180,E1 32892.204,E2 32892.204} C_VEL
LIN {X 0,Y 688.457,Z 335.479,A -85,B 0,C 180,E1 32889.181,E2 32889.181} C_VEL
LIN {X 0,Y 688.402,Z 335.482,A -85,B 0,C 180,E1 32886.343,E2 32886.343} C_VEL
LIN {X 0,Y 688.464,Z 335.6,A -85,B 0,C 180,E1 32885.695,E2 32885.695} C_VEL
LIN {X 0,Y 692.869,Z 347.981,A -85,B 0,C 180,E1 32884.401,E2 32884.401} C_VEL
LIN {X 0,Y 698.642,Z 358.523,A -85,B 0,C 180,E1 32883.919,E2 32883.919} C_VEL
LIN {X 0,Y 700.126,Z 364.887,A -85,B 0,C 180,E1 32883.752,E2 32883.752} C_VEL
LIN {X 0,Y 698.375,Z 600.807,A -85,B 0,C 180,E1 32880.973,E2 32880.973} C_VEL
LIN {X 0,Y 697.349,Z 737.279,A -85,B 0,C 180,E1 32879.374,E2 32879.374} C_VEL
LIN {X 0,Y 696.842,Z 762.859,A -85,B 0,C 180,E1 32878.926,E2 32878.926} C_VEL
LIN {X 0,Y 696.277,Z 784.6,A -85,B 0,C 180,E1 32878.407,E2 32878.407} C_VEL
LIN {X 0,Y 695.613,Z 809.119,A -85,B 0,C 180,E1 32877.664,E2 32877.664} C_VEL
LIN {X 0,Y 694.904,Z 829.549,A -85,B 0,C 180,E1 32876.906,E2 32876.906} C_VEL
LIN {X 0,Y 694.092,Z 852.08,A -85,B 0,C 180,E1 32875.926,E2 32875.926} C_VEL
LIN {X 0,Y 693.244,Z 873.505,A -85,B 0,C 180,E1 32874.817,E2 32874.817} C_VEL
LIN {X 0,Y 692.427,Z 893.68,A -85,B 0,C 180,E1 32873.623,E2 32873.623} C_VEL
LIN {X 0,Y 691.596,Z 913.623,A -85,B 0,C 180,E1 32872.259,E2 32872.259} C_VEL
LIN {X 0,Y 690.85,Z 932.283,A -85,B 0,C 180,E1 32870.813,E2 32870.813} C_VEL
LIN {X 0,Y 690.186,Z 949.438,A -85,B 0,C 180,E1 32869.288,E2 32869.288} C_VEL
LIN {X 0,Y 689.612,Z 965.236,A -85,B 0,C 180,E1 32867.71,E2 32867.71} C_VEL
LIN {X 0,Y 689.106,Z 980.853,A -85,B 0,C 180,E1 32865.917,E2 32865.917} C_VEL
LIN {X 0,Y 688.706,Z 994.67,A -85,B 0,C 180,E1 32864.109,E2 32864.109} C_VEL
LIN {X 0,Y 688.405,Z 1006.847,A -85,B 0,C 180,E1 32862.243,E2 32862.243} C_VEL
LIN {X 0,Y 688.205,Z 1017.368,A -85,B 0,C 180,E1 32860.379,E2 32860.379} C_VEL
LIN {X 0,Y 688.065,Z 1026.459,A -85,B 0,C 180,E1 32858.44,E2 32858.44} C_VEL
LIN {X 0,Y 687.961,Z 1033.322,A -85,B 0,C 180,E1 32856.677,E2 32856.677} C_VEL
LIN {X 0,Y 687.929,Z 1039.568,A -85,B 0,C 180,E1 32854.669,E2 32854.669} C_VEL
LIN {X 0,Y 687.911,Z 1043.735,A -85,B 0,C 180,E1 32852.833,E2 32852.833} C_VEL
LIN {X 0,Y 687.912,Z 1046.513,A -85,B 0,C 180,E1 32851.083,E2 32851.083} C_VEL
LIN {X 0,Y 687.913,Z 1048.226,A -85,B 0,C 180,E1 32849.001,E2 32849.001} C_VEL
LIN {X 0,Y 687.901,Z 1048.296,A -85,B 0,C 180,E1 32847.167,E2 32847.167} C_VEL
LIN {X 0,Y 687.899,Z 1046.967,A -85,B 0,C 180,E1 32845.164,E2 32845.164} C_VEL
LIN {X 0,Y 687.914,Z 1044.042,A -85,B 0,C 180,E1 32843.239,E2 32843.239} C_VEL
LIN {X 0,Y 687.924,Z 1040.142,A -85,B 0,C 180,E1 32841.474,E2 32841.474} C_VEL
LIN {X 0,Y 687.96,Z 1033.791,A -85,B 0,C 180,E1 32839.363,E2 32839.363} C_VEL
LIN {X 0,Y 688.058,Z 1026.922,A -85,B 0,C 180,E1 32837.58,E2 32837.58} C_VEL
LIN {X 0,Y 688.197,Z 1017.816,A -85,B 0,C 180,E1 32835.614,E2 32835.614} C_VEL
LIN {X 0,Y 688.398,Z 1007.167,A -85,B 0,C 180,E1 32833.72,E2 32833.72} C_VEL
LIN {X 0,Y 688.704,Z 994.743,A -85,B 0,C 180,E1 32831.811,E2 32831.811} C_VEL
LIN {X 0,Y 689.089,Z 981.417,A -85,B 0,C 180,E1 32830.063,E2 32830.063} C_VEL
LIN {X 0,Y 689.58,Z 966.197,A -85,B 0,C 180,E1 32828.3,E2 32828.3} C_VEL
LIN {X 0,Y 690.172,Z 949.803,A -85,B 0,C 180,E1 32826.657,E2 32826.657} C_VEL
LIN {X 0,Y 690.854,Z 932.213,A -85,B 0,C 180,E1 32825.091,E2 32825.091} C_VEL
LIN {X 0,Y 691.597,Z 913.611,A -85,B 0,C 180,E1 32823.65,E2 32823.65} C_VEL
LIN {X 0,Y 692.455,Z 893.015,A -85,B 0,C 180,E1 32822.246,E2 32822.246} C_VEL
LIN {X 0,Y 693.237,Z 873.73,A -85,B 0,C 180,E1 32821.105,E2 32821.105} C_VEL
LIN {X 0,Y 694.099,Z 851.82,A -85,B 0,C 180,E1 32819.972,E2 32819.972} C_VEL
LIN {X 0,Y 694.886,Z 830.038,A -85,B 0,C 180,E1 32819.023,E2 32819.023} C_VEL
LIN {X 0,Y 695.629,Z 808.789,A -85,B 0,C 180,E1 32818.234,E2 32818.234} C_VEL
LIN {X 0,Y 696.285,Z 784.259,A -85,B 0,C 180,E1 32817.494,E2 32817.494} C_VEL
LIN {X 0,Y 696.859,Z 762.366,A -85,B 0,C 180,E1 32816.974,E2 32816.974} C_VEL
LIN {X 0,Y 697.352,Z 737.001,A -85,B 0,C 180,E1 32816.532,E2 32816.532} C_VEL
LIN {X 0,Y 699.01,Z 511.807,A -85,B 0,C 180,E1 32813.896,E2 32813.896} C_VEL
LIN {X 0,Y 699.971,Z 363.45,A -85,B 0,C 180,E1 32812.131,E2 32812.131} C_VEL
LIN {X 0,Y 697.936,Z 356.872,A -85,B 0,C 180,E1 32811.928,E2 32811.928} C_VEL
LIN {X 0,Y 692.659,Z 347.51,A -85,B 0,C 180,E1 32811.482,E2 32811.482} C_VEL
LIN {X 0,Y 688.441,Z 335.478,A -85,B 0,C 180,E1 32810.17,E2 32810.17} C_VEL
LIN {X 0,Y 688.4,Z 335.479,A -85,B 0,C 180,E1 32807.401,E2 32807.401} C_VEL
LIN {X 0,Y 688.466,Z 335.473,A -85,B 0,C 180,E1 32804.512,E2 32804.512} C_VEL
LIN {X 0,Y 688.4,Z 335.47,A -85,B 0,C 180,E1 32801.58,E2 32801.58} C_VEL
LIN {X 0,Y 688.422,Z 335.474,A -85,B 0,C 180,E1 32798.863,E2 32798.863} C_VEL
LIN {X 0,Y 688.415,Z 335.457,A -85,B 0,C 180,E1 32795.716,E2 32795.716} C_VEL
LIN {X 0,Y 688.404,Z 335.476,A -85,B 0,C 180,E1 32793.003,E2 32793.003} C_VEL
LIN {X 0,Y 688.461,Z 335.471,A -85,B 0,C 180,E1 32789.974,E2 32789.974} C_VEL
LIN {X 0,Y 688.398,Z 335.475,A -85,B 0,C 180,E1 32787.135,E2 32787.135} C_VEL
LIN {X 0,Y 688.464,Z 335.474,A -85,B 0,C 180,E1 32784.269,E2 32784.269} C_VEL
LIN {X 0,Y 688.403,Z 335.47,A -85,B 0,C 180,E1 32781.292,E2 32781.292} C_VEL
LIN {X 0,Y 688.411,Z 335.476,A -85,B 0,C 180,E1 32778.635,E2 32778.635} C_VEL
LIN {X 0,Y 688.427,Z 335.471,A -85,B 0,C 180,E1 32775.501,E2 32775.501} C_VEL
LIN {X 0,Y 688.396,Z 335.473,A -85,B 0,C 180,E1 32772.84,E2 32772.84} C_VEL
LIN {X 0,Y 688.465,Z 335.47,A -85,B 0,C 180,E1 32769.952,E2 32769.952} C_VEL
LIN {X 0,Y 688.401,Z 335.473,A -85,B 0,C 180,E1 32767.008,E2 32767.008} C_VEL
LIN {X 0,Y 688.415,Z 335.474,A -85,B 0,C 180,E1 32764.332,E2 32764.332} C_VEL
LIN {X 0,Y 688.417,Z 335.468,A -85,B 0,C 180,E1 32761.165,E2 32761.165} C_VEL
LIN {X 0,Y 688.398,Z 335.475,A -85,B 0,C 180,E1 32758.502,E2 32758.502} C_VEL
LIN {X 0,Y 688.467,Z 335.474,A -85,B 0,C 180,E1 32755.585,E2 32755.585} C_VEL
LIN {X 0,Y 688.396,Z 335.467,A -85,B 0,C 180,E1 32752.74,E2 32752.74} C_VEL
LIN {X 0,Y 688.412,Z 335.477,A -85,B 0,C 180,E1 32750.131,E2 32750.131} C_VEL
LIN {X 0,Y 688.423,Z 335.472,A -85,B 0,C 180,E1 32746.99,E2 32746.99} C_VEL
LIN {X 0,Y 688.394,Z 335.469,A -85,B 0,C 180,E1 32744.326,E2 32744.326} C_VEL
LIN {X 0,Y 688.466,Z 335.469,A -85,B 0,C 180,E1 32741.454,E2 32741.454} C_VEL
LIN {X 0,Y 688.399,Z 335.474,A -85,B 0,C 180,E1 32738.529,E2 32738.529} C_VEL
LIN {X 0,Y 688.408,Z 335.471,A -85,B 0,C 180,E1 32735.912,E2 32735.912} C_VEL
LIN {X 0,Y 688.437,Z 335.469,A -85,B 0,C 180,E1 32732.867,E2 32732.867} C_VEL
LIN {X 0,Y 688.393,Z 335.474,A -85,B 0,C 180,E1 32730.214,E2 32730.214} C_VEL
LIN {X 0,Y 688.439,Z 335.478,A -85,B 0,C 180,E1 32727.494,E2 32727.494} C_VEL
LIN {X 0,Y 688.407,Z 335.474,A -85,B 0,C 180,E1 32724.428,E2 32724.428} C_VEL
LIN {X 0,Y 688.401,Z 335.476,A -85,B 0,C 180,E1 32721.774,E2 32721.774} C_VEL
LIN {X 0,Y 688.454,Z 335.472,A -85,B 0,C 180,E1 32718.747,E2 32718.747} C_VEL
LIN {X 0,Y 688.393,Z 335.476,A -85,B 0,C 180,E1 32715.913,E2 32715.913} C_VEL
LIN {X 0,Y 688.46,Z 335.472,A -85,B 0,C 180,E1 32713.048,E2 32713.048} C_VEL
LIN {X 0,Y 688.404,Z 335.481,A -85,B 0,C 180,E1 32710.158,E2 32710.158} C_VEL
LIN {X 0,Y 688.407,Z 335.577,A -85,B 0,C 180,E1 32709.887,E2 32709.887} C_VEL
LIN {X 0,Y 696.632,Z 357.318,A -85,B 0,C 180,E1 32707.694,E2 32707.694} C_VEL
LIN {X 0,Y 696.264,Z 377.414,A -85,B 0,C 180,E1 32706.245,E2 32706.245} C_VEL
LIN {X 0,Y 700.173,Z 394.081,A -85,B 0,C 180,E1 32705.804,E2 32705.804} C_VEL
LIN {X 0,Y 698.195,Z 655.721,A -85,B 0,C 180,E1 32702.729,E2 32702.729} C_VEL
LIN {X 0,Y 697.347,Z 767.4,A -85,B 0,C 180,E1 32701.417,E2 32701.417} C_VEL
LIN {X 0,Y 696.839,Z 792.889,A -85,B 0,C 180,E1 32700.97,E2 32700.97} C_VEL
LIN {X 0,Y 696.274,Z 814.669,A -85,B 0,C 180,E1 32700.45,E2 32700.45} C_VEL
LIN {X 0,Y 695.638,Z 838.557,A -85,B 0,C 180,E1 32699.729,E2 32699.729} C_VEL
LIN {X 0,Y 694.912,Z 859.353,A -85,B 0,C 180,E1 32698.959,E2 32698.959} C_VEL
LIN {X 0,Y 694.117,Z 881.251,A -85,B 0,C 180,E1 32698.009,E2 32698.009} C_VEL
LIN {X 0,Y 693.26,Z 903.137,A -85,B 0,C 180,E1 32696.882,E2 32696.882} C_VEL
LIN {X 0,Y 692.485,Z 922.179,A -85,B 0,C 180,E1 32695.761,E2 32695.761} C_VEL
LIN {X 0,Y 691.611,Z 943.23,A -85,B 0,C 180,E1 32694.333,E2 32694.333} C_VEL
LIN {X 0,Y 690.896,Z 961.056,A -85,B 0,C 180,E1 32692.956,E2 32692.956} C_VEL
LIN {X 0,Y 690.21,Z 978.605,A -85,B 0,C 180,E1 32691.412,E2 32691.412} C_VEL
LIN {X 0,Y 689.671,Z 993.638,A -85,B 0,C 180,E1 32689.92,E2 32689.92} C_VEL
LIN {X 0,Y 689.135,Z 1009.813,A -85,B 0,C 180,E1 32688.089,E2 32688.089} C_VEL
LIN {X 0,Y 688.749,Z 1022.529,A -85,B 0,C 180,E1 32686.445,E2 32686.445} C_VEL
LIN {X 0,Y 688.429,Z 1035.761,A -85,B 0,C 180,E1 32684.467,E2 32684.467} C_VEL
LIN {X 0,Y 688.229,Z 1045.568,A -85,B 0,C 180,E1 32682.758,E2 32682.758} C_VEL
LIN {X 0,Y 688.07,Z 1055.475,A -85,B 0,C 180,E1 32680.72,E2 32680.72} C_VEL
LIN {X 0,Y 687.974,Z 1062.513,A -85,B 0,C 180,E1 32678.947,E2 32678.947} C_VEL
LIN {X 0,Y 687.953,Z 1068.507,A -85,B 0,C 180,E1 32677.097,E2 32677.097} C_VEL
LIN {X 0,Y 687.923,Z 1073.497,A -85,B 0,C 180,E1 32675.003,E2 32675.003} C_VEL
LIN {X 0,Y 687.916,Z 1076.461,A -85,B 0,C 180,E1 32673.166,E2 32673.166} C_VEL
LIN {X 0,Y 687.914,Z 1078.239,A -85,B 0,C 180,E1 32670.999,E2 32670.999} C_VEL
LIN {X 0,Y 687.898,Z 1078.306,A -85,B 0,C 180,E1 32669.25,E2 32669.25} C_VEL
LIN {X 0,Y 687.907,Z 1077.017,A -85,B 0,C 180,E1 32667.251,E2 32667.251} C_VEL
LIN {X 0,Y 687.92,Z 1073.973,A -85,B 0,C 180,E1 32665.248,E2 32665.248} C_VEL
LIN {X 0,Y 687.916,Z 1070.07,A -85,B 0,C 180,E1 32663.49,E2 32663.49} C_VEL
LIN {X 0,Y 687.961,Z 1063.726,A -85,B 0,C 180,E1 32661.39,E2 32661.39} C_VEL
LIN {X 0,Y 688.057,Z 1056.895,A -85,B 0,C 180,E1 32659.619,E2 32659.619} C_VEL
LIN {X 0,Y 688.19,Z 1047.863,A -85,B 0,C 180,E1 32657.668,E2 32657.668} C_VEL
LIN {X 0,Y 688.386,Z 1037.323,A -85,B 0,C 180,E1 32655.79,E2 32655.79} C_VEL
LIN {X 0,Y 688.696,Z 1025.063,A -85,B 0,C 180,E1 32653.901,E2 32653.901} C_VEL
LIN {X 0,Y 689.094,Z 1011.228,A -85,B 0,C 180,E1 32652.084,E2 32652.084} C_VEL
LIN {X 0,Y 689.579,Z 996.173,A -85,B 0,C 180,E1 32650.342,E2 32650.342} C_VEL
LIN {X 0,Y 690.14,Z 980.462,A -85,B 0,C 180,E1 32648.764,E2 32648.764} C_VEL
LIN {X 0,Y 690.837,Z 962.713,A -85,B 0,C 180,E1 32647.177,E2 32647.177} C_VEL
LIN {X 0,Y 691.588,Z 943.837,A -85,B 0,C 180,E1 32645.712,E2 32645.712} C_VEL
LIN {X 0,Y 692.427,Z 923.628,A -85,B 0,C 180,E1 32644.329,E2 32644.329} C_VEL
LIN {X 0,Y 693.227,Z 903.944,A -85,B 0,C 180,E1 32643.163,E2 32643.163} C_VEL
LIN {X 0,Y 694.09,Z 882.148,A -85,B 0,C 180,E1 32642.032,E2 32642.032} C_VEL
LIN {X 0,Y 694.871,Z 860.488,A -85,B 0,C 180,E1 32641.086,E2 32641.086} C_VEL
LIN {X 0,Y 695.586,Z 839.842,A -85,B 0,C 180,E1 32640.316,E2 32640.316} C_VEL
LIN {X 0,Y 696.272,Z 814.781,A -85,B 0,C 180,E1 32639.552,E2 32639.552} C_VEL
LIN {X 0,Y 696.834,Z 793.024,A -85,B 0,C 180,E1 32639.033,E2 32639.033} C_VEL
LIN {X 0,Y 697.348,Z 767.543,A -85,B 0,C 180,E1 32638.585,E2 32638.585} C_VEL
LIN {X 0,Y 698.179,Z 657.887,A -85,B 0,C 180,E1 32637.296,E2 32637.296} C_VEL
LIN {X 0,Y 700.161,Z 395.556,A -85,B 0,C 180,E1 32634.213,E2 32634.213} C_VEL
LIN {X 0,Y 699.898,Z 392.055,A -85,B 0,C 180,E1 32634.154,E2 32634.154} C_VEL
LIN {X 0,Y 696.185,Z 376.671,A -85,B 0,C 180,E1 32633.72,E2 32633.72} C_VEL
LIN {X 0,Y 696.517,Z 357.059,A -85,B 0,C 180,E1 32632.279,E2 32632.279} C_VEL
LIN {X 0,Y 689.28,Z 338.267,A -85,B 0,C 180,E1 32630.38,E2 32630.38} C_VEL
LIN {X 0,Y 688.395,Z 335.489,A -85,B 0,C 180,E1 32630.078,E2 32630.078} C_VEL
LIN {X 0,Y 688.457,Z 335.476,A -85,B 0,C 180,E1 32627.293,E2 32627.293} C_VEL
LIN {X 0,Y 688.401,Z 335.479,A -85,B 0,C 180,E1 32624.319,E2 32624.319} C_VEL
LIN {X 0,Y 688.404,Z 335.476,A -85,B 0,C 180,E1 32621.701,E2 32621.701} C_VEL
LIN {X 0,Y 688.446,Z 335.478,A -85,B 0,C 180,E1 32618.648,E2 32618.648} C_VEL
LIN {X 0,Y 688.395,Z 335.476,A -85,B 0,C 180,E1 32615.856,E2 32615.856} C_VEL
LIN {X 0,Y 688.464,Z 335.47,A -85,B 0,C 180,E1 32613,E2 32613} C_VEL
LIN {X 0,Y 688.4,Z 335.475,A -85,B 0,C 180,E1 32610.04,E2 32610.04} C_VEL
LIN {X 0,Y 688.408,Z 335.468,A -85,B 0,C 180,E1 32607.415,E2 32607.415} C_VEL
LIN {X 0,Y 688.438,Z 335.472,A -85,B 0,C 180,E1 32604.361,E2 32604.361} C_VEL
LIN {X 0,Y 688.394,Z 335.474,A -85,B 0,C 180,E1 32601.628,E2 32601.628} C_VEL
LIN {X 0,Y 688.466,Z 335.466,A -85,B 0,C 180,E1 32598.75,E2 32598.75} C_VEL
LIN {X 0,Y 688.4,Z 335.473,A -85,B 0,C 180,E1 32595.76,E2 32595.76} C_VEL
LIN {X 0,Y 688.414,Z 335.469,A -85,B 0,C 180,E1 32593.096,E2 32593.096} C_VEL
LIN {X 0,Y 688.42,Z 335.469,A -85,B 0,C 180,E1 32589.953,E2 32589.953} C_VEL
LIN {X 0,Y 688.398,Z 335.474,A -85,B 0,C 180,E1 32587.26,E2 32587.26} C_VEL
LIN {X 0,Y 688.465,Z 335.467,A -85,B 0,C 180,E1 32584.331,E2 32584.331} C_VEL
LIN {X 0,Y 688.397,Z 335.474,A -85,B 0,C 180,E1 32581.415,E2 32581.415} C_VEL
LIN {X 0,Y 688.436,Z 335.462,A -85,B 0,C 180,E1 32578.668,E2 32578.668} C_VEL
LIN {X 0,Y 688.41,Z 335.473,A -85,B 0,C 180,E1 32575.585,E2 32575.585} C_VEL
LIN {X 0,Y 688.404,Z 335.469,A -85,B 0,C 180,E1 32572.908,E2 32572.908} C_VEL
LIN {X 0,Y 688.452,Z 335.47,A -85,B 0,C 180,E1 32569.878,E2 32569.878} C_VEL
LIN {X 0,Y 688.398,Z 335.474,A -85,B 0,C 180,E1 32567.063,E2 32567.063} C_VEL
LIN {X 0,Y 688.461,Z 335.468,A -85,B 0,C 180,E1 32564.241,E2 32564.241} C_VEL
LIN {X 0,Y 688.406,Z 335.476,A -85,B 0,C 180,E1 32561.264,E2 32561.264} C_VEL
LIN {X 0,Y 688.411,Z 335.466,A -85,B 0,C 180,E1 32558.595,E2 32558.595} C_VEL
LIN {X 0,Y 688.444,Z 335.471,A -85,B 0,C 180,E1 32555.548,E2 32555.548} C_VEL
LIN {X 0,Y 688.399,Z 335.474,A -85,B 0,C 180,E1 32552.772,E2 32552.772} C_VEL
LIN {X 0,Y 688.415,Z 335.473,A -85,B 0,C 180,E1 32552.444,E2 32552.444} C_VEL
LIN {X 0,Y 687.487,Z 335.597,A -85,B 0,C 180,E1 32551.803,E2 32551.803} C_VEL
LIN {X 0,Y 681.003,Z 336.394,A -85,B 0,C 180,E1 32549.96,E2 32549.96} C_VEL
LIN {X 0,Y 680.52,Z 336.461,A -85,B 0,C 180,E1 32549.539,E2 32549.539} C_VEL
LIN {X 0,Y 680.46,Z 336.458,A -85,B 0,C 180,E1 32546.731,E2 32546.731} C_VEL
LIN {X 0,Y 680.521,Z 336.46,A -85,B 0,C 180,E1 32543.9,E2 32543.9} C_VEL
LIN {X 0,Y 680.467,Z 336.463,A -85,B 0,C 180,E1 32540.882,E2 32540.882} C_VEL
LIN {X 0,Y 680.481,Z 336.464,A -85,B 0,C 180,E1 32538.156,E2 32538.156} C_VEL
LIN {X 0,Y 680.479,Z 336.453,A -85,B 0,C 180,E1 32534.973,E2 32534.973} C_VEL
LIN {X 0,Y 680.465,Z 336.461,A -85,B 0,C 180,E1 32532.299,E2 32532.299} C_VEL
LIN {X 0,Y 680.531,Z 336.465,A -85,B 0,C 180,E1 32529.39,E2 32529.39} C_VEL
LIN {X 0,Y 680.464,Z 336.472,A -85,B 0,C 180,E1 32526.507,E2 32526.507} C_VEL
LIN {X 0,Y 680.495,Z 336.659,A -85,B 0,C 180,E1 32526.148,E2 32526.148} C_VEL
LIN {X 0,Y 684.717,Z 348.244,A -85,B 0,C 180,E1 32524.906,E2 32524.906} C_VEL
LIN {X 0,Y 692.718,Z 362.495,A -85,B 0,C 180,E1 32524.227,E2 32524.227} C_VEL
LIN {X 0,Y 693.619,Z 366.874,A -85,B 0,C 180,E1 32524.116,E2 32524.116} C_VEL
LIN {X 0,Y 691.647,Z 602.962,A -85,B 0,C 180,E1 32521.31,E2 32521.31} C_VEL
LIN {X 0,Y 690.512,Z 737.314,A -85,B 0,C 180,E1 32519.721,E2 32519.721} C_VEL
LIN {X 0,Y 689.962,Z 762.768,A -85,B 0,C 180,E1 32519.271,E2 32519.271} C_VEL
LIN {X 0,Y 689.334,Z 784.408,A -85,B 0,C 180,E1 32518.752,E2 32518.752} C_VEL
LIN {X 0,Y 688.597,Z 808.779,A -85,B 0,C 180,E1 32518.01,E2 32518.01} C_VEL
LIN {X 0,Y 687.812,Z 829.079,A -85,B 0,C 180,E1 32517.253,E2 32517.253} C_VEL
LIN {X 0,Y 686.937,Z 850.775,A -85,B 0,C 180,E1 32516.306,E2 32516.306} C_VEL
LIN {X 0,Y 685.975,Z 872.371,A -85,B 0,C 180,E1 32515.19,E2 32515.19} C_VEL
LIN {X 0,Y 685.133,Z 891.237,A -85,B 0,C 180,E1 32514.073,E2 32514.073} C_VEL
LIN {X 0,Y 684.11,Z 912.774,A -85,B 0,C 180,E1 32512.606,E2 32512.606} C_VEL
LIN {X 0,Y 683.33,Z 930.395,A -85,B 0,C 180,E1 32511.235,E2 32511.235} C_VEL
LIN {X 0,Y 682.514,Z 948.792,A -85,B 0,C 180,E1 32509.602,E2 32509.602} C_VEL
LIN {X 0,Y 681.886,Z 964.475,A -85,B 0,C 180,E1 32508.023,E2 32508.023} C_VEL
LIN {X 0,Y 681.282,Z 980.36,A -85,B 0,C 180,E1 32506.192,E2 32506.192} C_VEL
LIN {X 0,Y 680.848,Z 993.532,A -85,B 0,C 180,E1 32504.457,E2 32504.457} C_VEL
LIN {X 0,Y 680.49,Z 1006.483,A -85,B 0,C 180,E1 32502.474,E2 32502.474} C_VEL
LIN {X 0,Y 680.261,Z 1016.589,A -85,B 0,C 180,E1 32500.673,E2 32500.673} C_VEL
LIN {X 0,Y 680.076,Z 1026.209,A -85,B 0,C 180,E1 32498.625,E2 32498.625} C_VEL
LIN {X 0,Y 679.984,Z 1032.805,A -85,B 0,C 180,E1 32496.925,E2 32496.925} C_VEL
LIN {X 0,Y 679.948,Z 1038.981,A -85,B 0,C 180,E1 32494.977,E2 32494.977} C_VEL
LIN {X 0,Y 679.915,Z 1043.623,A -85,B 0,C 180,E1 32492.95,E2 32492.95} C_VEL
LIN {X 0,Y 679.91,Z 1046.433,A -85,B 0,C 180,E1 32491.18,E2 32491.18} C_VEL
LIN {X 0,Y 679.913,Z 1048.21,A -85,B 0,C 180,E1 32489.073,E2 32489.073} C_VEL
LIN {X 0,Y 679.899,Z 1048.312,A -85,B 0,C 180,E1 32487.218,E2 32487.218} C_VEL
LIN {X 0,Y 679.898,Z 1047.036,A -85,B 0,C 180,E1 32485.191,E2 32485.191} C_VEL
LIN {X 0,Y 679.915,Z 1044.156,A -85,B 0,C 180,E1 32483.244,E2 32483.244} C_VEL
LIN {X 0,Y 679.926,Z 1040.289,A -85,B 0,C 180,E1 32481.458,E2 32481.458} C_VEL
LIN {X 0,Y 679.968,Z 1034.312,A -85,B 0,C 180,E1 32479.408,E2 32479.408} C_VEL
LIN {X 0,Y 680.075,Z 1027.177,A -85,B 0,C 180,E1 32477.518,E2 32477.518} C_VEL
LIN {X 0,Y 680.233,Z 1018.137,A -85,B 0,C 180,E1 32475.529,E2 32475.529} C_VEL
LIN {X 0,Y 680.46,Z 1007.539,A -85,B 0,C 180,E1 32473.613,E2 32473.613} C_VEL
LIN {X 0,Y 680.784,Z 995.77,A -85,B 0,C 180,E1 32471.77,E2 32471.77} C_VEL
LIN {X 0,Y 681.237,Z 981.917,A -85,B 0,C 180,E1 32469.912,E2 32469.912} C_VEL
LIN {X 0,Y 681.793,Z 966.772,A -85,B 0,C 180,E1 32468.13,E2 32468.13} C_VEL
LIN {X 0,Y 682.45,Z 950.464,A -85,B 0,C 180,E1 32466.469,E2 32466.469} C_VEL
LIN {X 0,Y 683.237,Z 932.67,A -85,B 0,C 180,E1 32464.859,E2 32464.859} C_VEL
LIN {X 0,Y 684.068,Z 913.872,A -85,B 0,C 180,E1 32463.385,E2 32463.385} C_VEL
LIN {X 0,Y 685.043,Z 893.323,A -85,B 0,C 180,E1 32461.966,E2 32461.966} C_VEL
LIN {X 0,Y 685.942,Z 873.257,A -85,B 0,C 180,E1 32460.769,E2 32460.769} C_VEL
LIN {X 0,Y 686.886,Z 852.005,A -85,B 0,C 180,E1 32459.66,E2 32459.66} C_VEL
LIN {X 0,Y 687.783,Z 829.798,A -85,B 0,C 180,E1 32458.686,E2 32458.686} C_VEL
LIN {X 0,Y 688.576,Z 809.336,A -85,B 0,C 180,E1 32457.92,E2 32457.92} C_VEL
LIN {X 0,Y 689.331,Z 784.564,A -85,B 0,C 180,E1 32457.162,E2 32457.162} C_VEL
LIN {X 0,Y 689.959,Z 762.87,A -85,B 0,C 180,E1 32456.641,E2 32456.641} C_VEL
LIN {X 0,Y 690.513,Z 737.402,A -85,B 0,C 180,E1 32456.191,E2 32456.191} C_VEL
LIN {X 0,Y 691.622,Z 606.026,A -85,B 0,C 180,E1 32454.636,E2 32454.636} C_VEL
LIN {X 0,Y 693.584,Z 370.527,A -85,B 0,C 180,E1 32451.837,E2 32451.837} C_VEL
LIN {X 0,Y 693.423,Z 365.152,A -85,B 0,C 180,E1 32451.76,E2 32451.76} C_VEL
LIN {X 0,Y 692.074,Z 361.063,A -85,B 0,C 180,E1 32451.626,E2 32451.626} C_VEL
LIN {X 0,Y 684.501,Z 347.835,A -85,B 0,C 180,E1 32450.98,E2 32450.98} C_VEL
LIN {X 0,Y 680.464,Z 336.47,A -85,B 0,C 180,E1 32449.718,E2 32449.718} C_VEL
LIN {X 0,Y 680.482,Z 336.466,A -85,B 0,C 180,E1 32447.016,E2 32447.016} C_VEL
LIN {X 0,Y 680.484,Z 336.46,A -85,B 0,C 180,E1 32443.912,E2 32443.912} C_VEL
LIN {X 0,Y 680.46,Z 336.458,A -85,B 0,C 180,E1 32441.206,E2 32441.206} C_VEL
LIN {X 0,Y 680.529,Z 336.462,A -85,B 0,C 180,E1 32438.317,E2 32438.317} C_VEL
LIN {X 0,Y 680.457,Z 336.446,A -85,B 0,C 180,E1 32435.359,E2 32435.359} C_VEL
LIN {X 0,Y 680.499,Z 336.467,A -85,B 0,C 180,E1 32432.633,E2 32432.633} C_VEL
LIN {X 0,Y 680.472,Z 336.462,A -85,B 0,C 180,E1 32429.554,E2 32429.554} C_VEL
LIN {X 0,Y 680.467,Z 336.465,A -85,B 0,C 180,E1 32426.882,E2 32426.882} C_VEL
LIN {X 0,Y 680.514,Z 336.461,A -85,B 0,C 180,E1 32423.833,E2 32423.833} C_VEL
LIN {X 0,Y 680.458,Z 336.46,A -85,B 0,C 180,E1 32421.011,E2 32421.011} C_VEL
LIN {X 0,Y 680.523,Z 336.459,A -85,B 0,C 180,E1 32418.149,E2 32418.149} C_VEL
LIN {X 0,Y 680.461,Z 336.462,A -85,B 0,C 180,E1 32415.163,E2 32415.163} C_VEL
LIN {X 0,Y 680.476,Z 336.464,A -85,B 0,C 180,E1 32412.474,E2 32412.474} C_VEL
LIN {X 0,Y 680.478,Z 336.459,A -85,B 0,C 180,E1 32409.302,E2 32409.302} C_VEL
LIN {X 0,Y 680.462,Z 336.464,A -85,B 0,C 180,E1 32406.581,E2 32406.581} C_VEL
LIN {X 0,Y 680.523,Z 336.461,A -85,B 0,C 180,E1 32403.622,E2 32403.622} C_VEL
LIN {X 0,Y 680.457,Z 336.459,A -85,B 0,C 180,E1 32400.758,E2 32400.758} C_VEL
LIN {X 0,Y 680.505,Z 336.465,A -85,B 0,C 180,E1 32397.979,E2 32397.979} C_VEL
LIN {X 0,Y 680.469,Z 336.462,A -85,B 0,C 180,E1 32394.942,E2 32394.942} C_VEL
LIN {X 0,Y 680.462,Z 336.458,A -85,B 0,C 180,E1 32392.315,E2 32392.315} C_VEL
LIN {X 0,Y 680.52,Z 336.453,A -85,B 0,C 180,E1 32389.331,E2 32389.331} C_VEL
LIN {X 0,Y 680.455,Z 336.464,A -85,B 0,C 180,E1 32386.488,E2 32386.488} C_VEL
LIN {X 0,Y 680.508,Z 336.459,A -85,B 0,C 180,E1 32383.701,E2 32383.701} C_VEL
LIN {X 0,Y 680.464,Z 336.455,A -85,B 0,C 180,E1 32380.693,E2 32380.693} C_VEL
LIN {X 0,Y 680.461,Z 336.465,A -85,B 0,C 180,E1 32378.085,E2 32378.085} C_VEL
LIN {X 0,Y 680.526,Z 336.461,A -85,B 0,C 180,E1 32375.152,E2 32375.152} C_VEL
LIN {X 0,Y 680.456,Z 336.461,A -85,B 0,C 180,E1 32372.237,E2 32372.237} C_VEL
LIN {X 0,Y 680.515,Z 336.466,A -85,B 0,C 180,E1 32369.431,E2 32369.431} C_VEL
LIN {X 0,Y 680.466,Z 336.464,A -85,B 0,C 180,E1 32366.425,E2 32366.425} C_VEL
LIN {X 0,Y 680.466,Z 336.467,A -85,B 0,C 180,E1 32363.776,E2 32363.776} C_VEL
LIN {X 0,Y 680.504,Z 336.463,A -85,B 0,C 180,E1 32360.707,E2 32360.707} C_VEL
LIN {X 0,Y 680.456,Z 336.465,A -85,B 0,C 180,E1 32357.928,E2 32357.928} C_VEL
LIN {X 0,Y 680.527,Z 336.463,A -85,B 0,C 180,E1 32355.03,E2 32355.03} C_VEL
LIN {X 0,Y 680.458,Z 336.468,A -85,B 0,C 180,E1 32352.072,E2 32352.072} C_VEL
LIN {X 0,Y 680.49,Z 336.536,A -85,B 0,C 180,E1 32350.349,E2 32350.349} C_VEL
LIN {X 0,Y 689.626,Z 360.874,A -85,B 0,C 180,E1 32347.857,E2 32347.857} C_VEL
